(* Schneider Machine Expert - Basic project 29Juli2020, file version 2.4.0.0 *)
(* ProjectInformations: Name=New project *)

HARDWARE
  Cpu 0: TM221CE16R
  ModuleExtensionObject 0: TM3AI8/G
  EthernetConfiguration: NetworkName=M221, IpAllocationMode=FixedAddress, IpAddress=192.168.10.91, SubnetMask=255.255.255.0
  SerialLineConfiguration: Baud=Baud19200, Parity=ParityEven, DataBits=DataBits8, StopBits=StopBits1, PhysicalMedium=PhysicalMediumRs485, TransmissionMode=TransmissionModeModbusRtu, SlaveId=1, Addressing=SlaveAddressing
  MastTask: UsePeriodScanMode=false, PeriodScan=100
  FastTask: Period=255
  CpuBehavior: StartingMode=StartAsPreviousState, AutoSaveRamOnEeprom=true, WatchdogPeriod=250

SYMBOLS  (address, symbol, comment, settings)
  %HSC0       [Type=SimpleCounter, Preset=0, UseDoubleWord=true, DedicatedInputs(DedicatedInput(Activated=true)), ReflexOutputs(ReflexOutput(Activated=false, LessThanS0=false, GreaterOrEqualThanS0=false, GreaterOrEqualThanS1=false), ReflexOutput(Activated=false, LessThanS0=false, GreaterOrEqualThanS0=false, GreaterOrEqualThanS1=false)), Thresholds(Threshold(ThresholdType=NotUsed, Priority=7), Threshold(Threshold]
  %HSC1       [Type=SimpleCounter, Preset=0, UseDoubleWord=true, DedicatedInputs(DedicatedInput(Activated=true)), ReflexOutputs(ReflexOutput(Activated=false, LessThanS0=false, GreaterOrEqualThanS0=false, GreaterOrEqualThanS1=false), ReflexOutput(Activated=false, LessThanS0=false, GreaterOrEqualThanS0=false, GreaterOrEqualThanS1=false)), Thresholds(Threshold(ThresholdType=NotUsed, Priority=7), Threshold(Threshold]
  %IW1.0      [Type=Type_4_20mA, Scope=Scope_Customized, Minimum=4000, Maximum=20000]
  %IW1.1      [Type=Type_4_20mA, Scope=Scope_Customized, Minimum=4000, Maximum=20000]
  %IW1.2      [Type=Type_4_20mA, Scope=Scope_Customized, Minimum=4000, Maximum=20000]
  %IW1.3      [Type=Type_4_20mA, Scope=Scope_Customized, Minimum=4000, Maximum=20000]
  %IW1.4      [Type=Type_4_20mA, Scope=Scope_Customized, Minimum=4000, Maximum=20000]
  %IW1.5      [Type=Type_4_20mA, Scope=Scope_Customized, Minimum=4000, Maximum=20000]
  %IW1.6      [Type=Type_4_20mA, Scope=Scope_Customized, Minimum=4000, Maximum=20000]

POU 4mikronA
  (* SectionNumber=1 *)

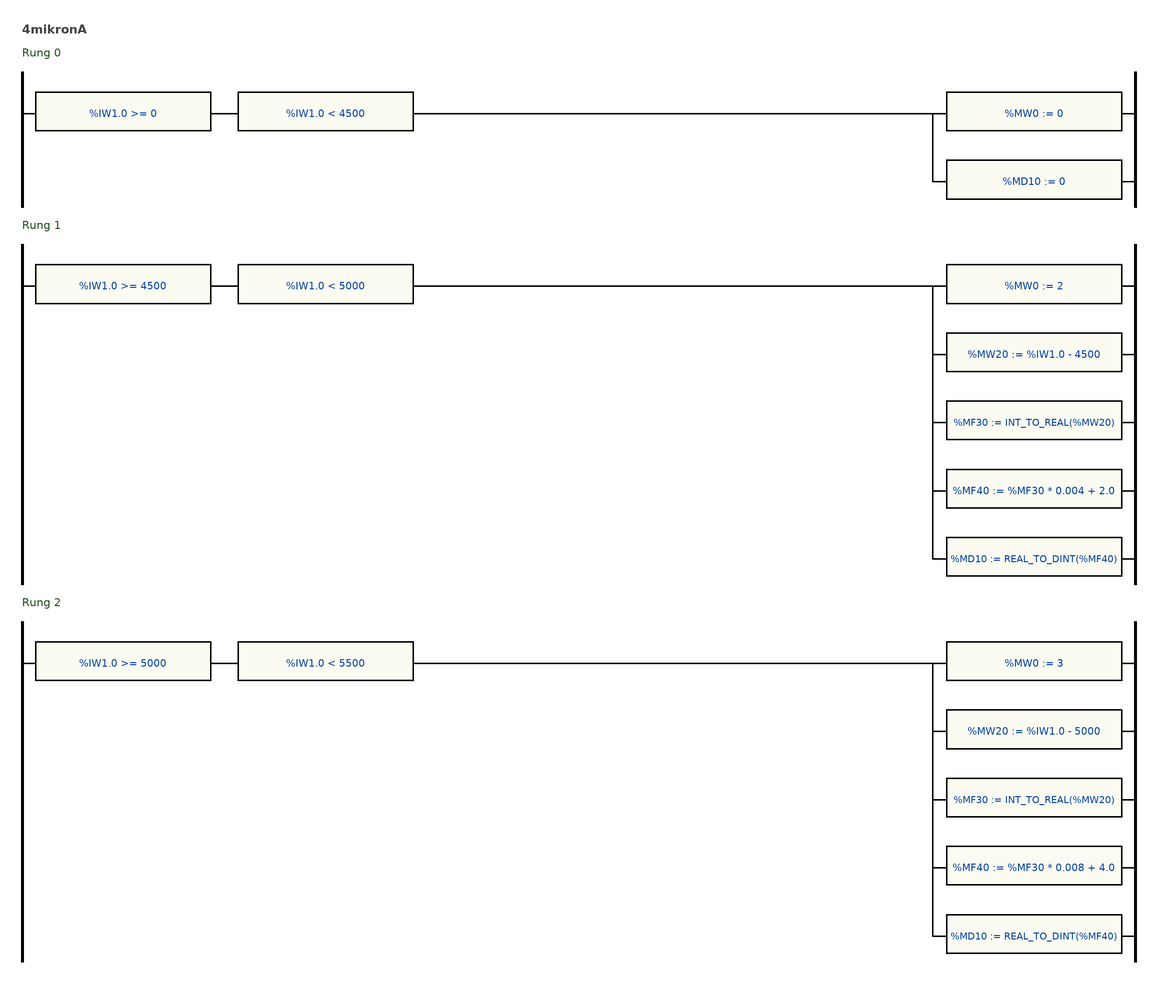

// Rung 0
  LD [ %IW1.0 >= 0 ]
  AND [ %IW1.0 < 4500 ]
  [ %MW0 := 0 ]
  [ %MD10 := 0 ]
  // as ST:
  //   IF %IW1.0 >= 0 AND %IW1.0 < 4500 THEN %MW0 := 0; END_IF;
  //   IF %IW1.0 >= 0 AND %IW1.0 < 4500 THEN %MD10 := 0; END_IF;

// Rung 1
  LD [ %IW1.0 >= 4500 ]
  AND [ %IW1.0 < 5000 ]
  [ %MW0 := 2 ]
  [ %MW20 := %IW1.0 - 4500 ]
  [ %MF30 := INT_TO_REAL ( %MW20 ) ]
  [ %MF40 := %MF30 * 0.004 + 2.0 ]
  [ %MD10 := REAL_TO_DINT ( %MF40 ) ]
  // as ST:
  //   IF %IW1.0 >= 4500 AND %IW1.0 < 5000 THEN %MW0 := 2; END_IF;
  //   IF %IW1.0 >= 4500 AND %IW1.0 < 5000 THEN %MW20 := %IW1.0 - 4500; END_IF;
  //   IF %IW1.0 >= 4500 AND %IW1.0 < 5000 THEN %MF30 := INT_TO_REAL ( %MW20 ); END_IF;
  //   IF %IW1.0 >= 4500 AND %IW1.0 < 5000 THEN %MF40 := %MF30 * 0.004 + 2.0; END_IF;
  //   IF %IW1.0 >= 4500 AND %IW1.0 < 5000 THEN %MD10 := REAL_TO_DINT ( %MF40 ); END_IF;

// Rung 2
  LD [ %IW1.0 >= 5000 ]
  AND [ %IW1.0 < 5500 ]
  [ %MW0 := 3 ]
  [ %MW20 := %IW1.0 - 5000 ]
  [ %MF30 := INT_TO_REAL ( %MW20 ) ]
  [ %MF40 := %MF30 * 0.008 + 4.0 ]
  [ %MD10 := REAL_TO_DINT ( %MF40 ) ]
  // as ST:
  //   IF %IW1.0 >= 5000 AND %IW1.0 < 5500 THEN %MW0 := 3; END_IF;
  //   IF %IW1.0 >= 5000 AND %IW1.0 < 5500 THEN %MW20 := %IW1.0 - 5000; END_IF;
  //   IF %IW1.0 >= 5000 AND %IW1.0 < 5500 THEN %MF30 := INT_TO_REAL ( %MW20 ); END_IF;
  //   IF %IW1.0 >= 5000 AND %IW1.0 < 5500 THEN %MF40 := %MF30 * 0.008 + 4.0; END_IF;
  //   IF %IW1.0 >= 5000 AND %IW1.0 < 5500 THEN %MD10 := REAL_TO_DINT ( %MF40 ); END_IF;

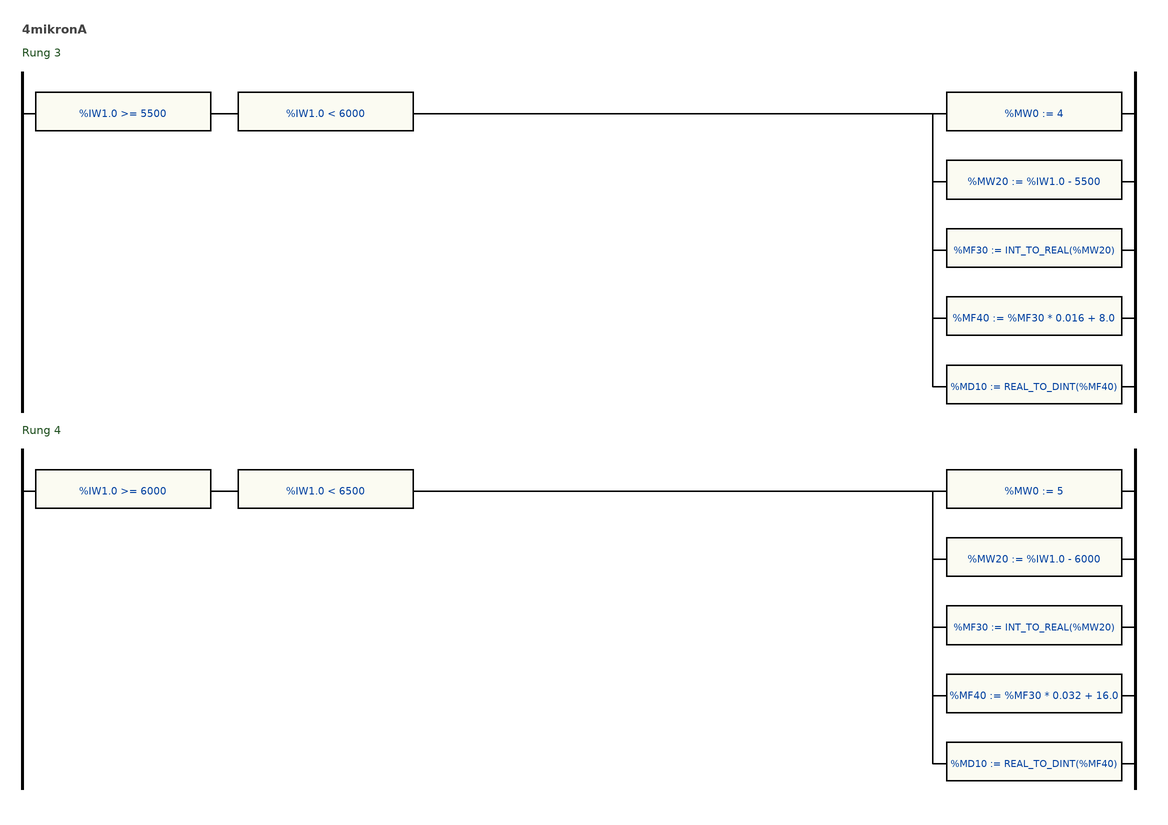

// Rung 3
  LD [ %IW1.0 >= 5500 ]
  AND [ %IW1.0 < 6000 ]
  [ %MW0 := 4 ]
  [ %MW20 := %IW1.0 - 5500 ]
  [ %MF30 := INT_TO_REAL ( %MW20 ) ]
  [ %MF40 := %MF30 * 0.016 + 8.0 ]
  [ %MD10 := REAL_TO_DINT ( %MF40 ) ]
  // as ST:
  //   IF %IW1.0 >= 5500 AND %IW1.0 < 6000 THEN %MW0 := 4; END_IF;
  //   IF %IW1.0 >= 5500 AND %IW1.0 < 6000 THEN %MW20 := %IW1.0 - 5500; END_IF;
  //   IF %IW1.0 >= 5500 AND %IW1.0 < 6000 THEN %MF30 := INT_TO_REAL ( %MW20 ); END_IF;
  //   IF %IW1.0 >= 5500 AND %IW1.0 < 6000 THEN %MF40 := %MF30 * 0.016 + 8.0; END_IF;
  //   IF %IW1.0 >= 5500 AND %IW1.0 < 6000 THEN %MD10 := REAL_TO_DINT ( %MF40 ); END_IF;

// Rung 4
  LD [ %IW1.0 >= 6000 ]
  AND [ %IW1.0 < 6500 ]
  [ %MW0 := 5 ]
  [ %MW20 := %IW1.0 - 6000 ]
  [ %MF30 := INT_TO_REAL ( %MW20 ) ]
  [ %MF40 := %MF30 * 0.032 + 16.0 ]
  [ %MD10 := REAL_TO_DINT ( %MF40 ) ]
  // as ST:
  //   IF %IW1.0 >= 6000 AND %IW1.0 < 6500 THEN %MW0 := 5; END_IF;
  //   IF %IW1.0 >= 6000 AND %IW1.0 < 6500 THEN %MW20 := %IW1.0 - 6000; END_IF;
  //   IF %IW1.0 >= 6000 AND %IW1.0 < 6500 THEN %MF30 := INT_TO_REAL ( %MW20 ); END_IF;
  //   IF %IW1.0 >= 6000 AND %IW1.0 < 6500 THEN %MF40 := %MF30 * 0.032 + 16.0; END_IF;
  //   IF %IW1.0 >= 6000 AND %IW1.0 < 6500 THEN %MD10 := REAL_TO_DINT ( %MF40 ); END_IF;

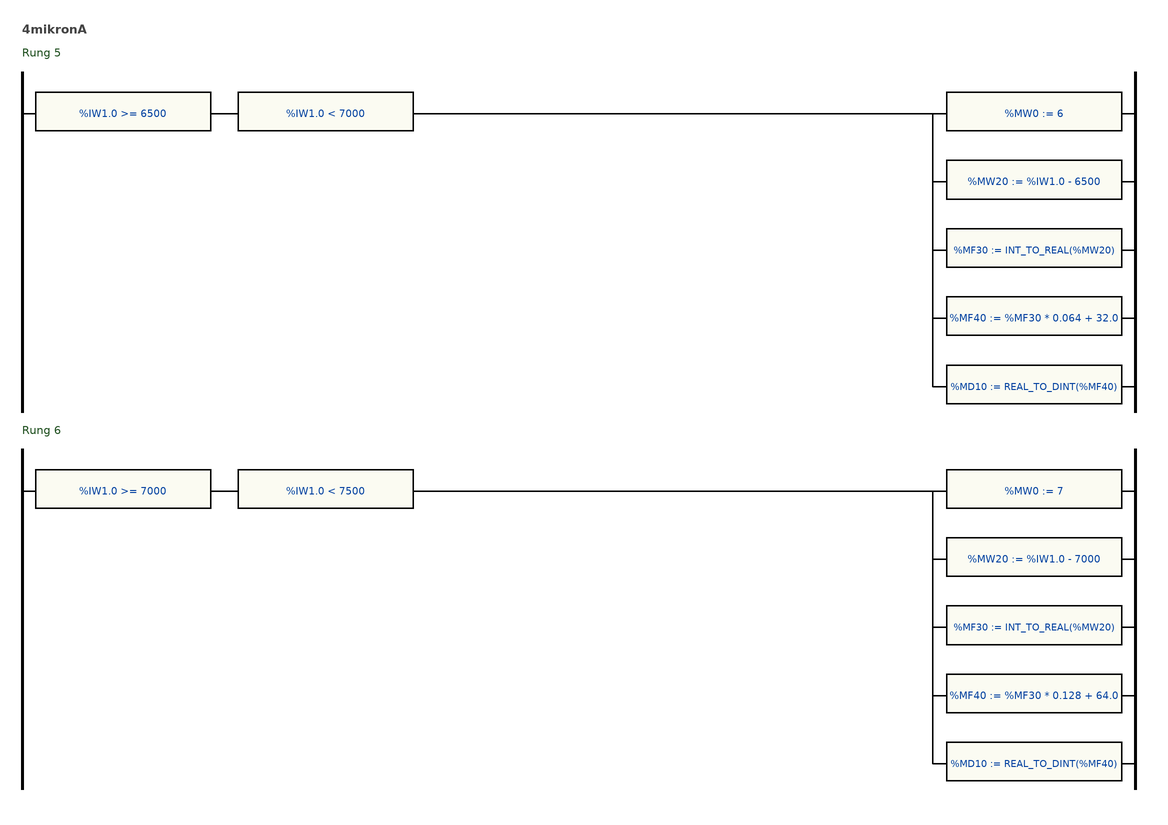

// Rung 5
  LD [ %IW1.0 >= 6500 ]
  AND [ %IW1.0 < 7000 ]
  [ %MW0 := 6 ]
  [ %MW20 := %IW1.0 - 6500 ]
  [ %MF30 := INT_TO_REAL ( %MW20 ) ]
  [ %MF40 := %MF30 * 0.064 + 32.0 ]
  [ %MD10 := REAL_TO_DINT ( %MF40 ) ]
  // as ST:
  //   IF %IW1.0 >= 6500 AND %IW1.0 < 7000 THEN %MW0 := 6; END_IF;
  //   IF %IW1.0 >= 6500 AND %IW1.0 < 7000 THEN %MW20 := %IW1.0 - 6500; END_IF;
  //   IF %IW1.0 >= 6500 AND %IW1.0 < 7000 THEN %MF30 := INT_TO_REAL ( %MW20 ); END_IF;
  //   IF %IW1.0 >= 6500 AND %IW1.0 < 7000 THEN %MF40 := %MF30 * 0.064 + 32.0; END_IF;
  //   IF %IW1.0 >= 6500 AND %IW1.0 < 7000 THEN %MD10 := REAL_TO_DINT ( %MF40 ); END_IF;

// Rung 6
  LD [ %IW1.0 >= 7000 ]
  AND [ %IW1.0 < 7500 ]
  [ %MW0 := 7 ]
  [ %MW20 := %IW1.0 - 7000 ]
  [ %MF30 := INT_TO_REAL ( %MW20 ) ]
  [ %MF40 := %MF30 * 0.128 + 64.0 ]
  [ %MD10 := REAL_TO_DINT ( %MF40 ) ]
  // as ST:
  //   IF %IW1.0 >= 7000 AND %IW1.0 < 7500 THEN %MW0 := 7; END_IF;
  //   IF %IW1.0 >= 7000 AND %IW1.0 < 7500 THEN %MW20 := %IW1.0 - 7000; END_IF;
  //   IF %IW1.0 >= 7000 AND %IW1.0 < 7500 THEN %MF30 := INT_TO_REAL ( %MW20 ); END_IF;
  //   IF %IW1.0 >= 7000 AND %IW1.0 < 7500 THEN %MF40 := %MF30 * 0.128 + 64.0; END_IF;
  //   IF %IW1.0 >= 7000 AND %IW1.0 < 7500 THEN %MD10 := REAL_TO_DINT ( %MF40 ); END_IF;

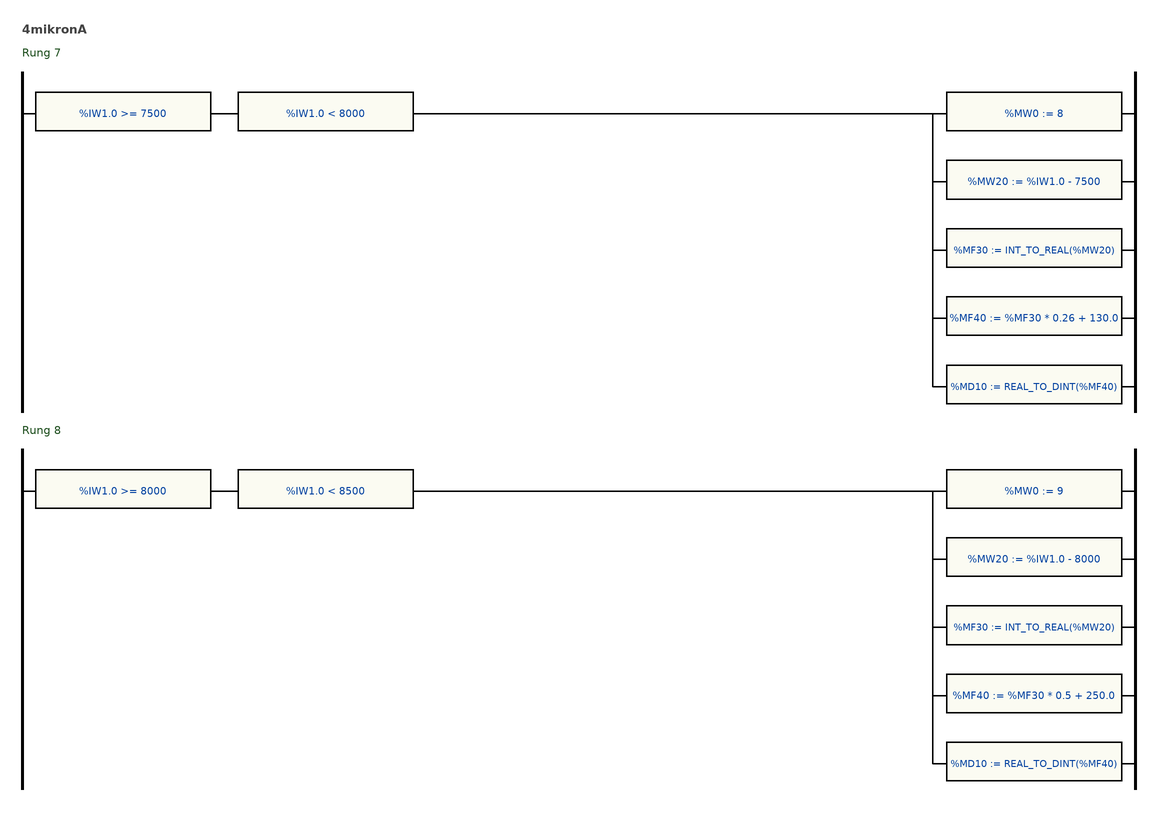

// Rung 7
  LD [ %IW1.0 >= 7500 ]
  AND [ %IW1.0 < 8000 ]
  [ %MW0 := 8 ]
  [ %MW20 := %IW1.0 - 7500 ]
  [ %MF30 := INT_TO_REAL ( %MW20 ) ]
  [ %MF40 := %MF30 * 0.26 + 130.0 ]
  [ %MD10 := REAL_TO_DINT ( %MF40 ) ]
  // as ST:
  //   IF %IW1.0 >= 7500 AND %IW1.0 < 8000 THEN %MW0 := 8; END_IF;
  //   IF %IW1.0 >= 7500 AND %IW1.0 < 8000 THEN %MW20 := %IW1.0 - 7500; END_IF;
  //   IF %IW1.0 >= 7500 AND %IW1.0 < 8000 THEN %MF30 := INT_TO_REAL ( %MW20 ); END_IF;
  //   IF %IW1.0 >= 7500 AND %IW1.0 < 8000 THEN %MF40 := %MF30 * 0.26 + 130.0; END_IF;
  //   IF %IW1.0 >= 7500 AND %IW1.0 < 8000 THEN %MD10 := REAL_TO_DINT ( %MF40 ); END_IF;

// Rung 8
  LD [ %IW1.0 >= 8000 ]
  AND [ %IW1.0 < 8500 ]
  [ %MW0 := 9 ]
  [ %MW20 := %IW1.0 - 8000 ]
  [ %MF30 := INT_TO_REAL ( %MW20 ) ]
  [ %MF40 := %MF30 * 0.5 + 250.0 ]
  [ %MD10 := REAL_TO_DINT ( %MF40 ) ]
  // as ST:
  //   IF %IW1.0 >= 8000 AND %IW1.0 < 8500 THEN %MW0 := 9; END_IF;
  //   IF %IW1.0 >= 8000 AND %IW1.0 < 8500 THEN %MW20 := %IW1.0 - 8000; END_IF;
  //   IF %IW1.0 >= 8000 AND %IW1.0 < 8500 THEN %MF30 := INT_TO_REAL ( %MW20 ); END_IF;
  //   IF %IW1.0 >= 8000 AND %IW1.0 < 8500 THEN %MF40 := %MF30 * 0.5 + 250.0; END_IF;
  //   IF %IW1.0 >= 8000 AND %IW1.0 < 8500 THEN %MD10 := REAL_TO_DINT ( %MF40 ); END_IF;

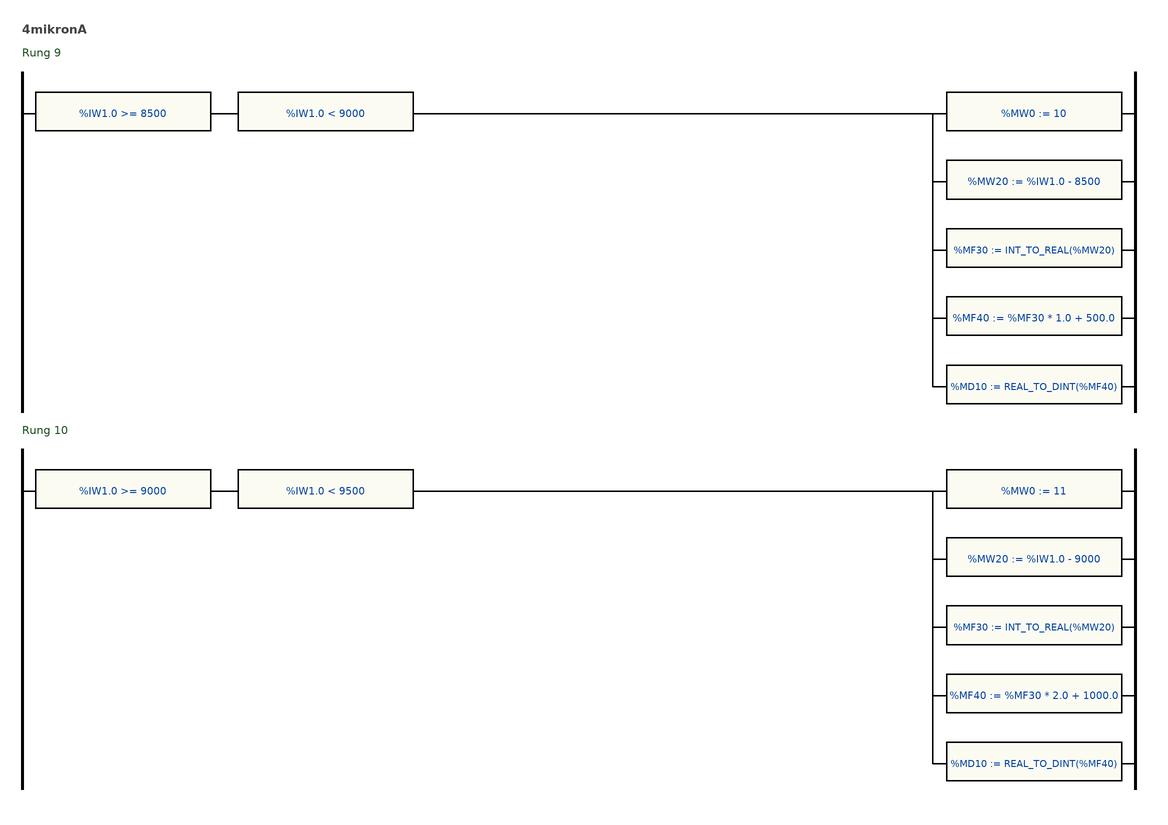

// Rung 9
  LD [ %IW1.0 >= 8500 ]
  AND [ %IW1.0 < 9000 ]
  [ %MW0 := 10 ]
  [ %MW20 := %IW1.0 - 8500 ]
  [ %MF30 := INT_TO_REAL ( %MW20 ) ]
  [ %MF40 := %MF30 * 1.0 + 500.0 ]
  [ %MD10 := REAL_TO_DINT ( %MF40 ) ]
  // as ST:
  //   IF %IW1.0 >= 8500 AND %IW1.0 < 9000 THEN %MW0 := 10; END_IF;
  //   IF %IW1.0 >= 8500 AND %IW1.0 < 9000 THEN %MW20 := %IW1.0 - 8500; END_IF;
  //   IF %IW1.0 >= 8500 AND %IW1.0 < 9000 THEN %MF30 := INT_TO_REAL ( %MW20 ); END_IF;
  //   IF %IW1.0 >= 8500 AND %IW1.0 < 9000 THEN %MF40 := %MF30 * 1.0 + 500.0; END_IF;
  //   IF %IW1.0 >= 8500 AND %IW1.0 < 9000 THEN %MD10 := REAL_TO_DINT ( %MF40 ); END_IF;

// Rung 10
  LD [ %IW1.0 >= 9000 ]
  AND [ %IW1.0 < 9500 ]
  [ %MW0 := 11 ]
  [ %MW20 := %IW1.0 - 9000 ]
  [ %MF30 := INT_TO_REAL ( %MW20 ) ]
  [ %MF40 := %MF30 * 2.0 + 1000.0 ]
  [ %MD10 := REAL_TO_DINT ( %MF40 ) ]
  // as ST:
  //   IF %IW1.0 >= 9000 AND %IW1.0 < 9500 THEN %MW0 := 11; END_IF;
  //   IF %IW1.0 >= 9000 AND %IW1.0 < 9500 THEN %MW20 := %IW1.0 - 9000; END_IF;
  //   IF %IW1.0 >= 9000 AND %IW1.0 < 9500 THEN %MF30 := INT_TO_REAL ( %MW20 ); END_IF;
  //   IF %IW1.0 >= 9000 AND %IW1.0 < 9500 THEN %MF40 := %MF30 * 2.0 + 1000.0; END_IF;
  //   IF %IW1.0 >= 9000 AND %IW1.0 < 9500 THEN %MD10 := REAL_TO_DINT ( %MF40 ); END_IF;

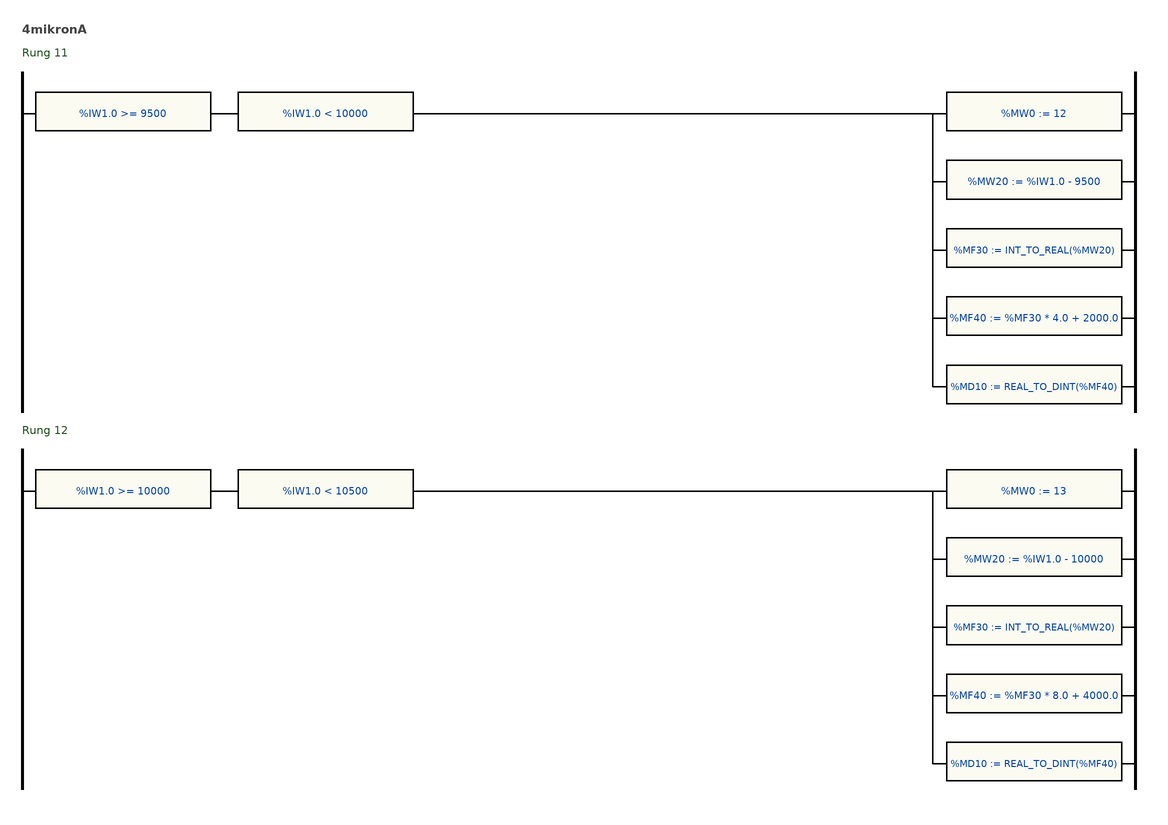

// Rung 11
  LD [ %IW1.0 >= 9500 ]
  AND [ %IW1.0 < 10000 ]
  [ %MW0 := 12 ]
  [ %MW20 := %IW1.0 - 9500 ]
  [ %MF30 := INT_TO_REAL ( %MW20 ) ]
  [ %MF40 := %MF30 * 4.0 + 2000.0 ]
  [ %MD10 := REAL_TO_DINT ( %MF40 ) ]
  // as ST:
  //   IF %IW1.0 >= 9500 AND %IW1.0 < 10000 THEN %MW0 := 12; END_IF;
  //   IF %IW1.0 >= 9500 AND %IW1.0 < 10000 THEN %MW20 := %IW1.0 - 9500; END_IF;
  //   IF %IW1.0 >= 9500 AND %IW1.0 < 10000 THEN %MF30 := INT_TO_REAL ( %MW20 ); END_IF;
  //   IF %IW1.0 >= 9500 AND %IW1.0 < 10000 THEN %MF40 := %MF30 * 4.0 + 2000.0; END_IF;
  //   IF %IW1.0 >= 9500 AND %IW1.0 < 10000 THEN %MD10 := REAL_TO_DINT ( %MF40 ); END_IF;

// Rung 12
  LD [ %IW1.0 >= 10000 ]
  AND [ %IW1.0 < 10500 ]
  [ %MW0 := 13 ]
  [ %MW20 := %IW1.0 - 10000 ]
  [ %MF30 := INT_TO_REAL ( %MW20 ) ]
  [ %MF40 := %MF30 * 8.0 + 4000.0 ]
  [ %MD10 := REAL_TO_DINT ( %MF40 ) ]
  // as ST:
  //   IF %IW1.0 >= 10000 AND %IW1.0 < 10500 THEN %MW0 := 13; END_IF;
  //   IF %IW1.0 >= 10000 AND %IW1.0 < 10500 THEN %MW20 := %IW1.0 - 10000; END_IF;
  //   IF %IW1.0 >= 10000 AND %IW1.0 < 10500 THEN %MF30 := INT_TO_REAL ( %MW20 ); END_IF;
  //   IF %IW1.0 >= 10000 AND %IW1.0 < 10500 THEN %MF40 := %MF30 * 8.0 + 4000.0; END_IF;
  //   IF %IW1.0 >= 10000 AND %IW1.0 < 10500 THEN %MD10 := REAL_TO_DINT ( %MF40 ); END_IF;

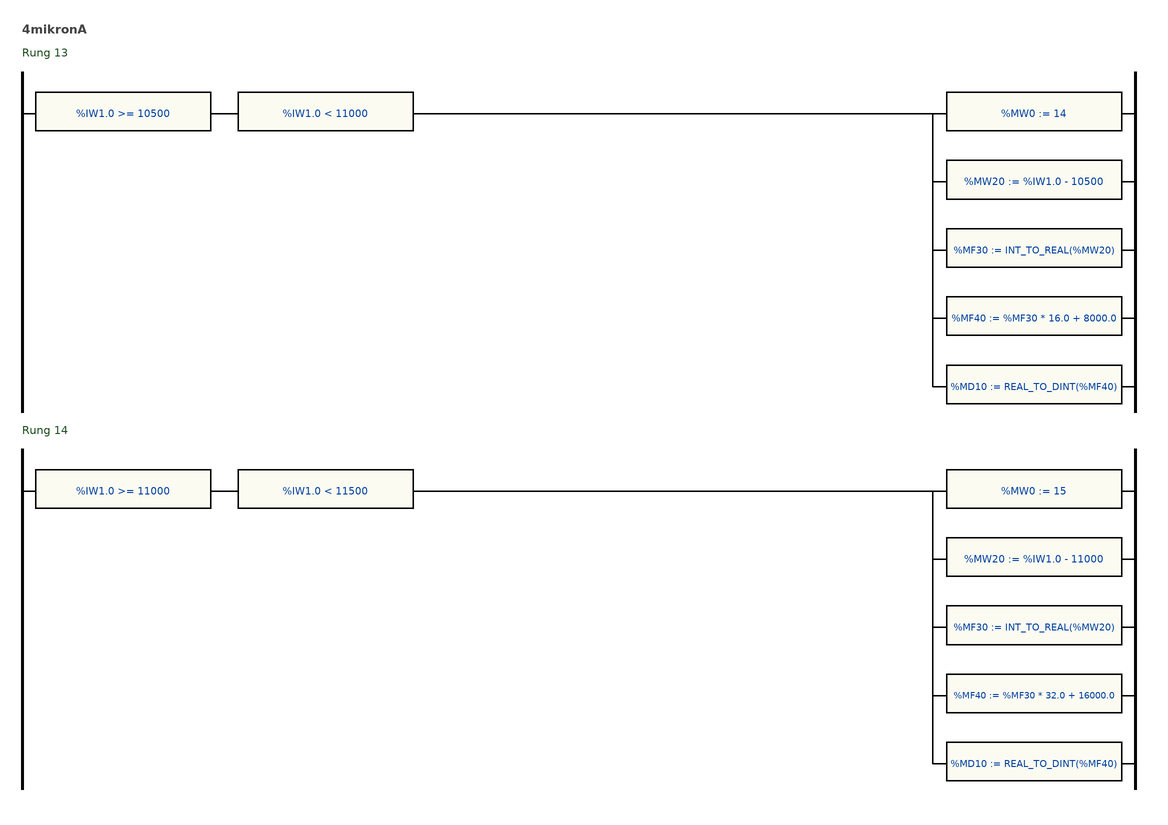

// Rung 13
  LD [ %IW1.0 >= 10500 ]
  AND [ %IW1.0 < 11000 ]
  [ %MW0 := 14 ]
  [ %MW20 := %IW1.0 - 10500 ]
  [ %MF30 := INT_TO_REAL ( %MW20 ) ]
  [ %MF40 := %MF30 * 16.0 + 8000.0 ]
  [ %MD10 := REAL_TO_DINT ( %MF40 ) ]
  // as ST:
  //   IF %IW1.0 >= 10500 AND %IW1.0 < 11000 THEN %MW0 := 14; END_IF;
  //   IF %IW1.0 >= 10500 AND %IW1.0 < 11000 THEN %MW20 := %IW1.0 - 10500; END_IF;
  //   IF %IW1.0 >= 10500 AND %IW1.0 < 11000 THEN %MF30 := INT_TO_REAL ( %MW20 ); END_IF;
  //   IF %IW1.0 >= 10500 AND %IW1.0 < 11000 THEN %MF40 := %MF30 * 16.0 + 8000.0; END_IF;
  //   IF %IW1.0 >= 10500 AND %IW1.0 < 11000 THEN %MD10 := REAL_TO_DINT ( %MF40 ); END_IF;

// Rung 14
  LD [ %IW1.0 >= 11000 ]
  AND [ %IW1.0 < 11500 ]
  [ %MW0 := 15 ]
  [ %MW20 := %IW1.0 - 11000 ]
  [ %MF30 := INT_TO_REAL ( %MW20 ) ]
  [ %MF40 := %MF30 * 32.0 + 16000.0 ]
  [ %MD10 := REAL_TO_DINT ( %MF40 ) ]
  // as ST:
  //   IF %IW1.0 >= 11000 AND %IW1.0 < 11500 THEN %MW0 := 15; END_IF;
  //   IF %IW1.0 >= 11000 AND %IW1.0 < 11500 THEN %MW20 := %IW1.0 - 11000; END_IF;
  //   IF %IW1.0 >= 11000 AND %IW1.0 < 11500 THEN %MF30 := INT_TO_REAL ( %MW20 ); END_IF;
  //   IF %IW1.0 >= 11000 AND %IW1.0 < 11500 THEN %MF40 := %MF30 * 32.0 + 16000.0; END_IF;
  //   IF %IW1.0 >= 11000 AND %IW1.0 < 11500 THEN %MD10 := REAL_TO_DINT ( %MF40 ); END_IF;

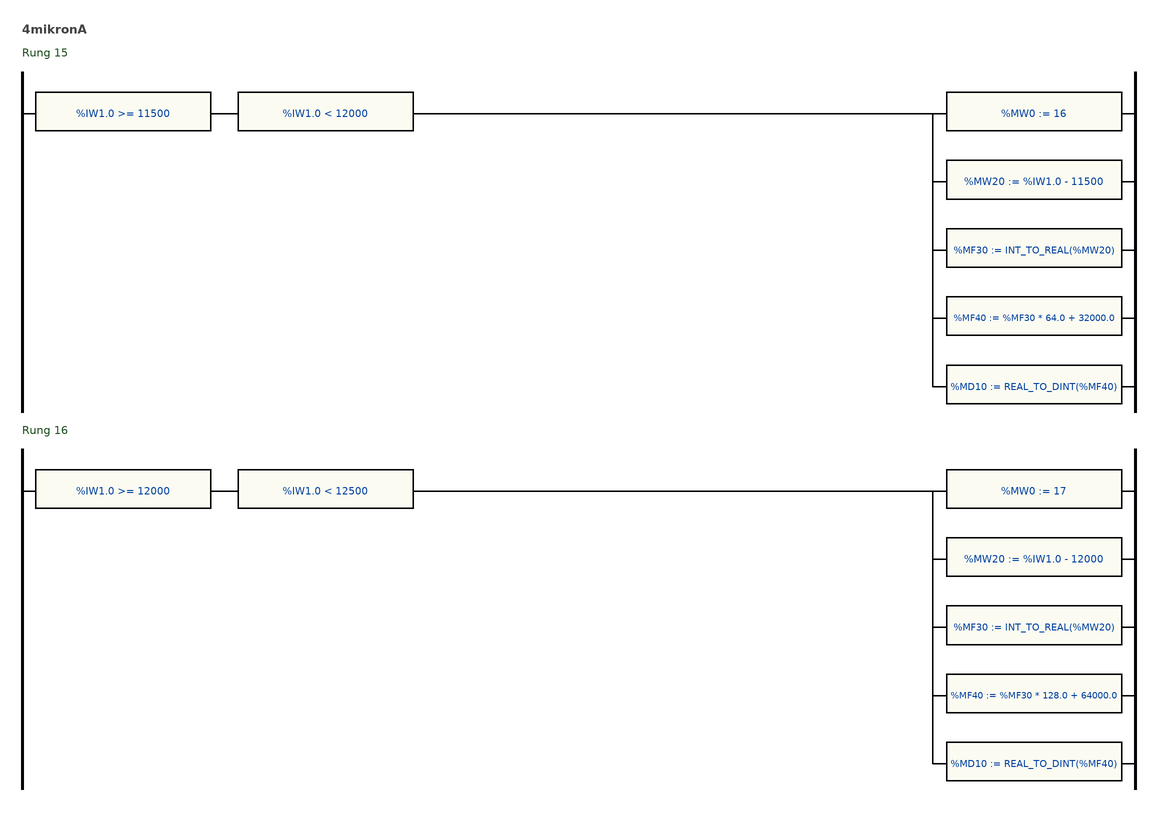

// Rung 15
  LD [ %IW1.0 >= 11500 ]
  AND [ %IW1.0 < 12000 ]
  [ %MW0 := 16 ]
  [ %MW20 := %IW1.0 - 11500 ]
  [ %MF30 := INT_TO_REAL ( %MW20 ) ]
  [ %MF40 := %MF30 * 64.0 + 32000.0 ]
  [ %MD10 := REAL_TO_DINT ( %MF40 ) ]
  // as ST:
  //   IF %IW1.0 >= 11500 AND %IW1.0 < 12000 THEN %MW0 := 16; END_IF;
  //   IF %IW1.0 >= 11500 AND %IW1.0 < 12000 THEN %MW20 := %IW1.0 - 11500; END_IF;
  //   IF %IW1.0 >= 11500 AND %IW1.0 < 12000 THEN %MF30 := INT_TO_REAL ( %MW20 ); END_IF;
  //   IF %IW1.0 >= 11500 AND %IW1.0 < 12000 THEN %MF40 := %MF30 * 64.0 + 32000.0; END_IF;
  //   IF %IW1.0 >= 11500 AND %IW1.0 < 12000 THEN %MD10 := REAL_TO_DINT ( %MF40 ); END_IF;

// Rung 16
  LD [ %IW1.0 >= 12000 ]
  AND [ %IW1.0 < 12500 ]
  [ %MW0 := 17 ]
  [ %MW20 := %IW1.0 - 12000 ]
  [ %MF30 := INT_TO_REAL ( %MW20 ) ]
  [ %MF40 := %MF30 * 128.0 + 64000.0 ]
  [ %MD10 := REAL_TO_DINT ( %MF40 ) ]
  // as ST:
  //   IF %IW1.0 >= 12000 AND %IW1.0 < 12500 THEN %MW0 := 17; END_IF;
  //   IF %IW1.0 >= 12000 AND %IW1.0 < 12500 THEN %MW20 := %IW1.0 - 12000; END_IF;
  //   IF %IW1.0 >= 12000 AND %IW1.0 < 12500 THEN %MF30 := INT_TO_REAL ( %MW20 ); END_IF;
  //   IF %IW1.0 >= 12000 AND %IW1.0 < 12500 THEN %MF40 := %MF30 * 128.0 + 64000.0; END_IF;
  //   IF %IW1.0 >= 12000 AND %IW1.0 < 12500 THEN %MD10 := REAL_TO_DINT ( %MF40 ); END_IF;

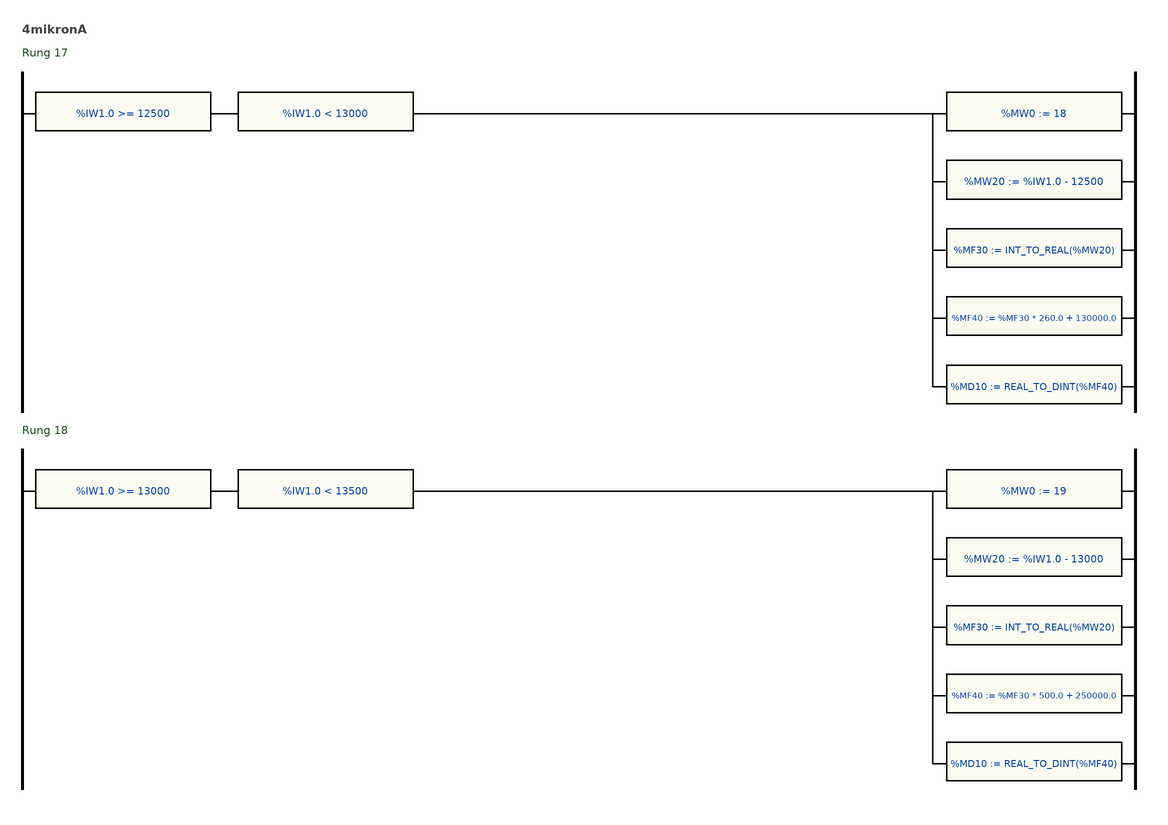

// Rung 17
  LD [ %IW1.0 >= 12500 ]
  AND [ %IW1.0 < 13000 ]
  [ %MW0 := 18 ]
  [ %MW20 := %IW1.0 - 12500 ]
  [ %MF30 := INT_TO_REAL ( %MW20 ) ]
  [ %MF40 := %MF30 * 260.0 + 130000.0 ]
  [ %MD10 := REAL_TO_DINT ( %MF40 ) ]
  // as ST:
  //   IF %IW1.0 >= 12500 AND %IW1.0 < 13000 THEN %MW0 := 18; END_IF;
  //   IF %IW1.0 >= 12500 AND %IW1.0 < 13000 THEN %MW20 := %IW1.0 - 12500; END_IF;
  //   IF %IW1.0 >= 12500 AND %IW1.0 < 13000 THEN %MF30 := INT_TO_REAL ( %MW20 ); END_IF;
  //   IF %IW1.0 >= 12500 AND %IW1.0 < 13000 THEN %MF40 := %MF30 * 260.0 + 130000.0; END_IF;
  //   IF %IW1.0 >= 12500 AND %IW1.0 < 13000 THEN %MD10 := REAL_TO_DINT ( %MF40 ); END_IF;

// Rung 18
  LD [ %IW1.0 >= 13000 ]
  AND [ %IW1.0 < 13500 ]
  [ %MW0 := 19 ]
  [ %MW20 := %IW1.0 - 13000 ]
  [ %MF30 := INT_TO_REAL ( %MW20 ) ]
  [ %MF40 := %MF30 * 500.0 + 250000.0 ]
  [ %MD10 := REAL_TO_DINT ( %MF40 ) ]
  // as ST:
  //   IF %IW1.0 >= 13000 AND %IW1.0 < 13500 THEN %MW0 := 19; END_IF;
  //   IF %IW1.0 >= 13000 AND %IW1.0 < 13500 THEN %MW20 := %IW1.0 - 13000; END_IF;
  //   IF %IW1.0 >= 13000 AND %IW1.0 < 13500 THEN %MF30 := INT_TO_REAL ( %MW20 ); END_IF;
  //   IF %IW1.0 >= 13000 AND %IW1.0 < 13500 THEN %MF40 := %MF30 * 500.0 + 250000.0; END_IF;
  //   IF %IW1.0 >= 13000 AND %IW1.0 < 13500 THEN %MD10 := REAL_TO_DINT ( %MF40 ); END_IF;

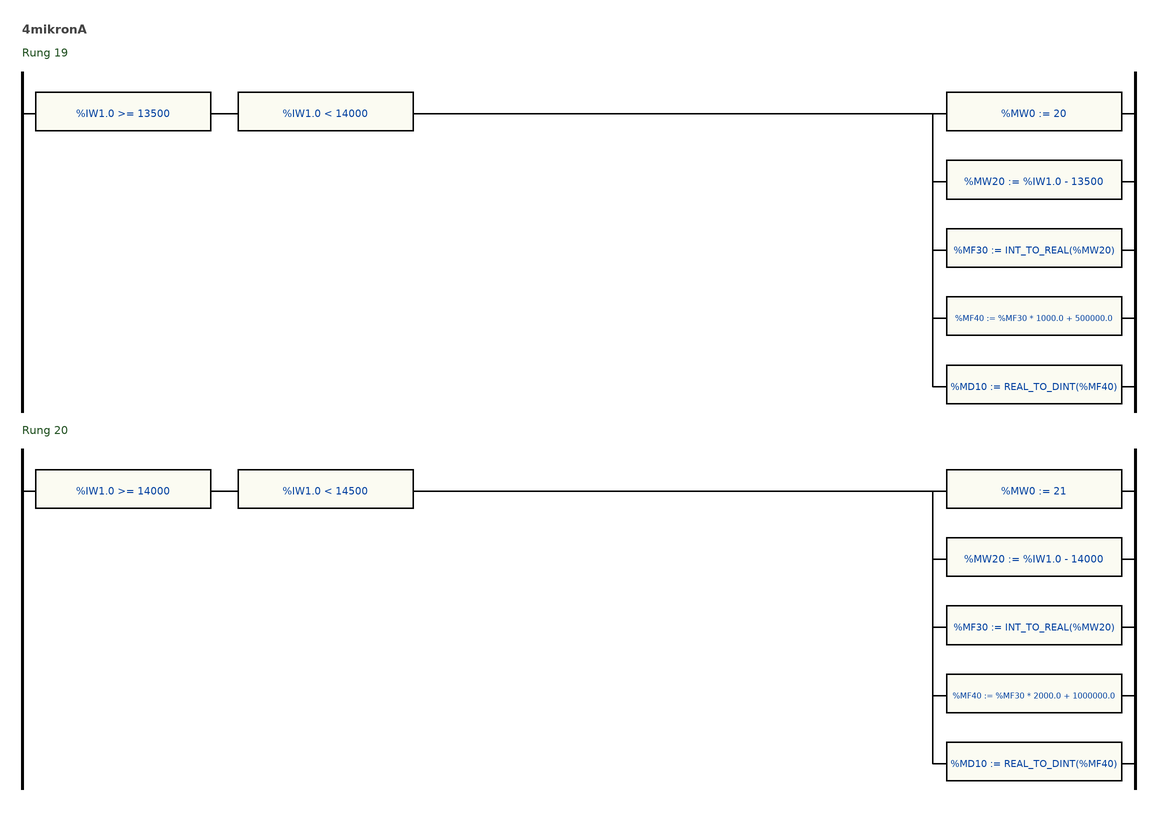

// Rung 19
  LD [ %IW1.0 >= 13500 ]
  AND [ %IW1.0 < 14000 ]
  [ %MW0 := 20 ]
  [ %MW20 := %IW1.0 - 13500 ]
  [ %MF30 := INT_TO_REAL ( %MW20 ) ]
  [ %MF40 := %MF30 * 1000.0 + 500000.0 ]
  [ %MD10 := REAL_TO_DINT ( %MF40 ) ]
  // as ST:
  //   IF %IW1.0 >= 13500 AND %IW1.0 < 14000 THEN %MW0 := 20; END_IF;
  //   IF %IW1.0 >= 13500 AND %IW1.0 < 14000 THEN %MW20 := %IW1.0 - 13500; END_IF;
  //   IF %IW1.0 >= 13500 AND %IW1.0 < 14000 THEN %MF30 := INT_TO_REAL ( %MW20 ); END_IF;
  //   IF %IW1.0 >= 13500 AND %IW1.0 < 14000 THEN %MF40 := %MF30 * 1000.0 + 500000.0; END_IF;
  //   IF %IW1.0 >= 13500 AND %IW1.0 < 14000 THEN %MD10 := REAL_TO_DINT ( %MF40 ); END_IF;

// Rung 20
  LD [ %IW1.0 >= 14000 ]
  AND [ %IW1.0 < 14500 ]
  [ %MW0 := 21 ]
  [ %MW20 := %IW1.0 - 14000 ]
  [ %MF30 := INT_TO_REAL ( %MW20 ) ]
  [ %MF40 := %MF30 * 2000.0 + 1000000.0 ]
  [ %MD10 := REAL_TO_DINT ( %MF40 ) ]
  // as ST:
  //   IF %IW1.0 >= 14000 AND %IW1.0 < 14500 THEN %MW0 := 21; END_IF;
  //   IF %IW1.0 >= 14000 AND %IW1.0 < 14500 THEN %MW20 := %IW1.0 - 14000; END_IF;
  //   IF %IW1.0 >= 14000 AND %IW1.0 < 14500 THEN %MF30 := INT_TO_REAL ( %MW20 ); END_IF;
  //   IF %IW1.0 >= 14000 AND %IW1.0 < 14500 THEN %MF40 := %MF30 * 2000.0 + 1000000.0; END_IF;
  //   IF %IW1.0 >= 14000 AND %IW1.0 < 14500 THEN %MD10 := REAL_TO_DINT ( %MF40 ); END_IF;

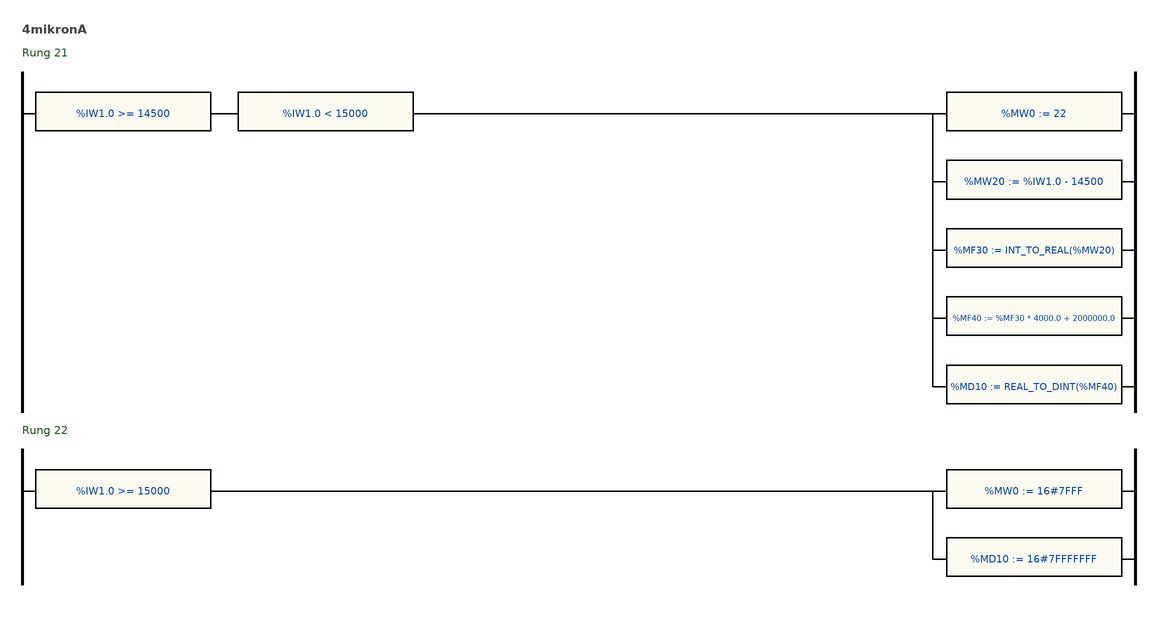

// Rung 21
  LD [ %IW1.0 >= 14500 ]
  AND [ %IW1.0 < 15000 ]
  [ %MW0 := 22 ]
  [ %MW20 := %IW1.0 - 14500 ]
  [ %MF30 := INT_TO_REAL ( %MW20 ) ]
  [ %MF40 := %MF30 * 4000.0 + 2000000.0 ]
  [ %MD10 := REAL_TO_DINT ( %MF40 ) ]
  // as ST:
  //   IF %IW1.0 >= 14500 AND %IW1.0 < 15000 THEN %MW0 := 22; END_IF;
  //   IF %IW1.0 >= 14500 AND %IW1.0 < 15000 THEN %MW20 := %IW1.0 - 14500; END_IF;
  //   IF %IW1.0 >= 14500 AND %IW1.0 < 15000 THEN %MF30 := INT_TO_REAL ( %MW20 ); END_IF;
  //   IF %IW1.0 >= 14500 AND %IW1.0 < 15000 THEN %MF40 := %MF30 * 4000.0 + 2000000.0; END_IF;
  //   IF %IW1.0 >= 14500 AND %IW1.0 < 15000 THEN %MD10 := REAL_TO_DINT ( %MF40 ); END_IF;

// Rung 22
  LD [ %IW1.0 >= 15000 ]
  [ %MW0 := 16#7FFF ]
  [ %MD10 := 16#7FFFFFFF ]
  // as ST:
  //   IF %IW1.0 >= 15000 THEN %MW0 := 16#7FFF; END_IF;
  //   IF %IW1.0 >= 15000 THEN %MD10 := 16#7FFFFFFF; END_IF;

POU 6mikronA
  (* SectionNumber=2 *)

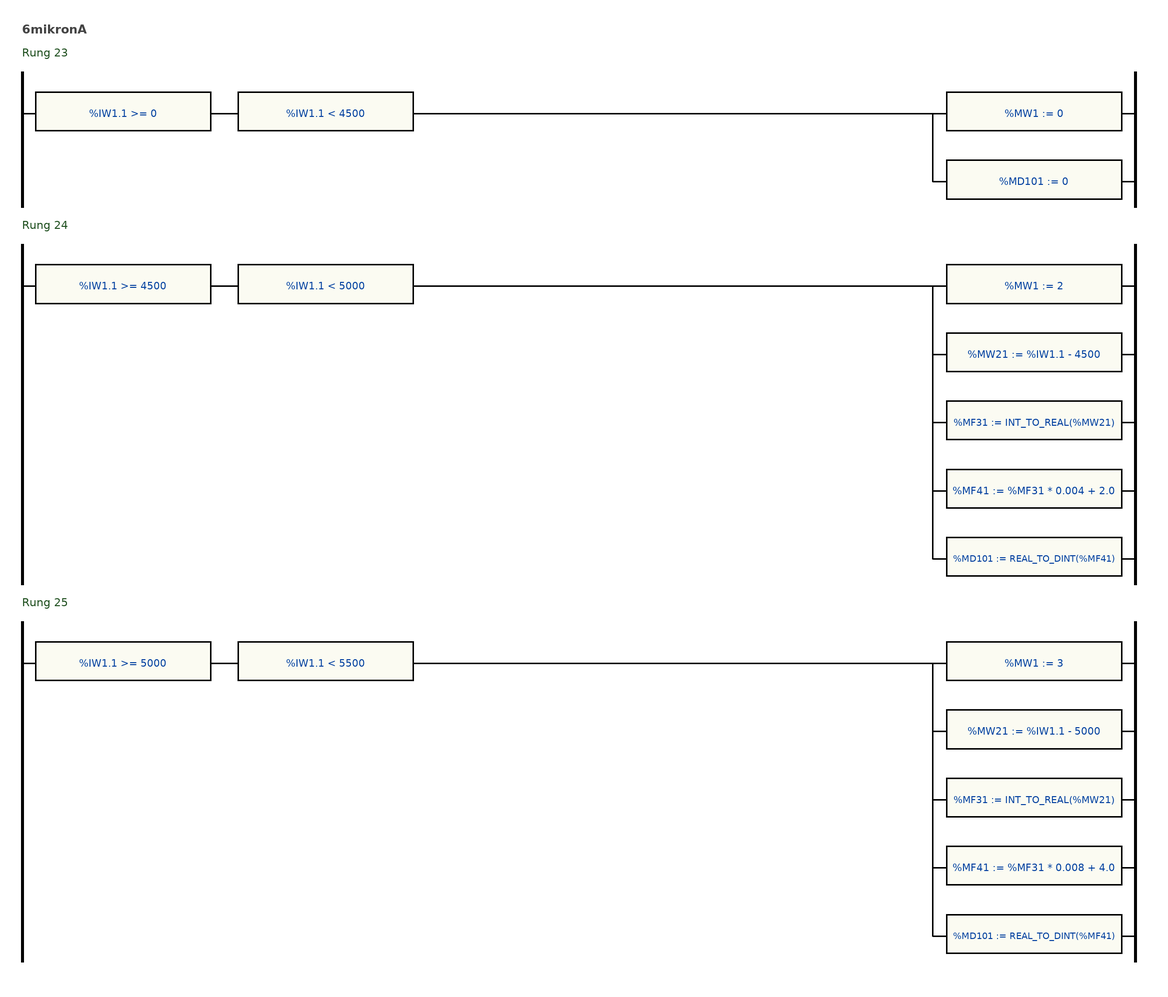

// Rung 23
  LD [ %IW1.1 >= 0 ]
  AND [ %IW1.1 < 4500 ]
  [ %MW1 := 0 ]
  [ %MD101 := 0 ]
  // as ST:
  //   IF %IW1.1 >= 0 AND %IW1.1 < 4500 THEN %MW1 := 0; END_IF;
  //   IF %IW1.1 >= 0 AND %IW1.1 < 4500 THEN %MD101 := 0; END_IF;

// Rung 24
  LD [ %IW1.1 >= 4500 ]
  AND [ %IW1.1 < 5000 ]
  [ %MW1 := 2 ]
  [ %MW21 := %IW1.1 - 4500 ]
  [ %MF31 := INT_TO_REAL ( %MW21 ) ]
  [ %MF41 := %MF31 * 0.004 + 2.0 ]
  [ %MD101 := REAL_TO_DINT ( %MF41 ) ]
  // as ST:
  //   IF %IW1.1 >= 4500 AND %IW1.1 < 5000 THEN %MW1 := 2; END_IF;
  //   IF %IW1.1 >= 4500 AND %IW1.1 < 5000 THEN %MW21 := %IW1.1 - 4500; END_IF;
  //   IF %IW1.1 >= 4500 AND %IW1.1 < 5000 THEN %MF31 := INT_TO_REAL ( %MW21 ); END_IF;
  //   IF %IW1.1 >= 4500 AND %IW1.1 < 5000 THEN %MF41 := %MF31 * 0.004 + 2.0; END_IF;
  //   IF %IW1.1 >= 4500 AND %IW1.1 < 5000 THEN %MD101 := REAL_TO_DINT ( %MF41 ); END_IF;

// Rung 25
  LD [ %IW1.1 >= 5000 ]
  AND [ %IW1.1 < 5500 ]
  [ %MW1 := 3 ]
  [ %MW21 := %IW1.1 - 5000 ]
  [ %MF31 := INT_TO_REAL ( %MW21 ) ]
  [ %MF41 := %MF31 * 0.008 + 4.0 ]
  [ %MD101 := REAL_TO_DINT ( %MF41 ) ]
  // as ST:
  //   IF %IW1.1 >= 5000 AND %IW1.1 < 5500 THEN %MW1 := 3; END_IF;
  //   IF %IW1.1 >= 5000 AND %IW1.1 < 5500 THEN %MW21 := %IW1.1 - 5000; END_IF;
  //   IF %IW1.1 >= 5000 AND %IW1.1 < 5500 THEN %MF31 := INT_TO_REAL ( %MW21 ); END_IF;
  //   IF %IW1.1 >= 5000 AND %IW1.1 < 5500 THEN %MF41 := %MF31 * 0.008 + 4.0; END_IF;
  //   IF %IW1.1 >= 5000 AND %IW1.1 < 5500 THEN %MD101 := REAL_TO_DINT ( %MF41 ); END_IF;

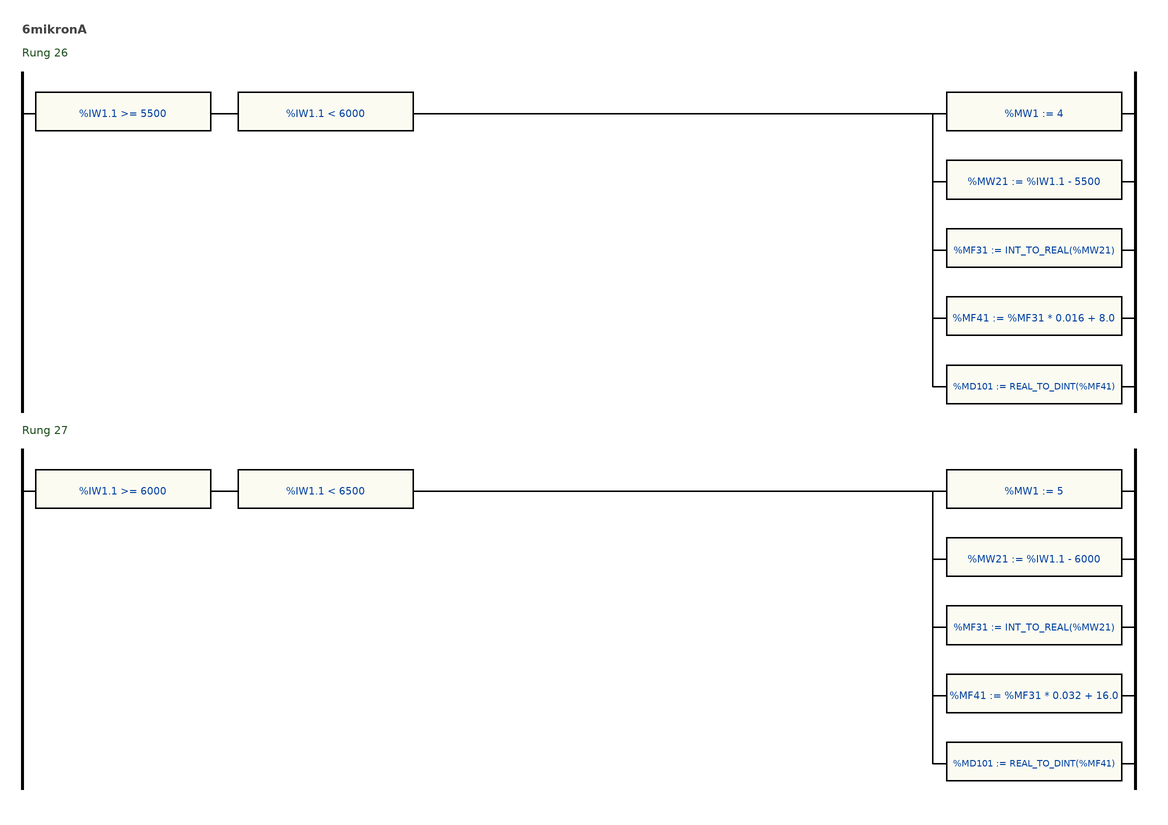

// Rung 26
  LD [ %IW1.1 >= 5500 ]
  AND [ %IW1.1 < 6000 ]
  [ %MW1 := 4 ]
  [ %MW21 := %IW1.1 - 5500 ]
  [ %MF31 := INT_TO_REAL ( %MW21 ) ]
  [ %MF41 := %MF31 * 0.016 + 8.0 ]
  [ %MD101 := REAL_TO_DINT ( %MF41 ) ]
  // as ST:
  //   IF %IW1.1 >= 5500 AND %IW1.1 < 6000 THEN %MW1 := 4; END_IF;
  //   IF %IW1.1 >= 5500 AND %IW1.1 < 6000 THEN %MW21 := %IW1.1 - 5500; END_IF;
  //   IF %IW1.1 >= 5500 AND %IW1.1 < 6000 THEN %MF31 := INT_TO_REAL ( %MW21 ); END_IF;
  //   IF %IW1.1 >= 5500 AND %IW1.1 < 6000 THEN %MF41 := %MF31 * 0.016 + 8.0; END_IF;
  //   IF %IW1.1 >= 5500 AND %IW1.1 < 6000 THEN %MD101 := REAL_TO_DINT ( %MF41 ); END_IF;

// Rung 27
  LD [ %IW1.1 >= 6000 ]
  AND [ %IW1.1 < 6500 ]
  [ %MW1 := 5 ]
  [ %MW21 := %IW1.1 - 6000 ]
  [ %MF31 := INT_TO_REAL ( %MW21 ) ]
  [ %MF41 := %MF31 * 0.032 + 16.0 ]
  [ %MD101 := REAL_TO_DINT ( %MF41 ) ]
  // as ST:
  //   IF %IW1.1 >= 6000 AND %IW1.1 < 6500 THEN %MW1 := 5; END_IF;
  //   IF %IW1.1 >= 6000 AND %IW1.1 < 6500 THEN %MW21 := %IW1.1 - 6000; END_IF;
  //   IF %IW1.1 >= 6000 AND %IW1.1 < 6500 THEN %MF31 := INT_TO_REAL ( %MW21 ); END_IF;
  //   IF %IW1.1 >= 6000 AND %IW1.1 < 6500 THEN %MF41 := %MF31 * 0.032 + 16.0; END_IF;
  //   IF %IW1.1 >= 6000 AND %IW1.1 < 6500 THEN %MD101 := REAL_TO_DINT ( %MF41 ); END_IF;

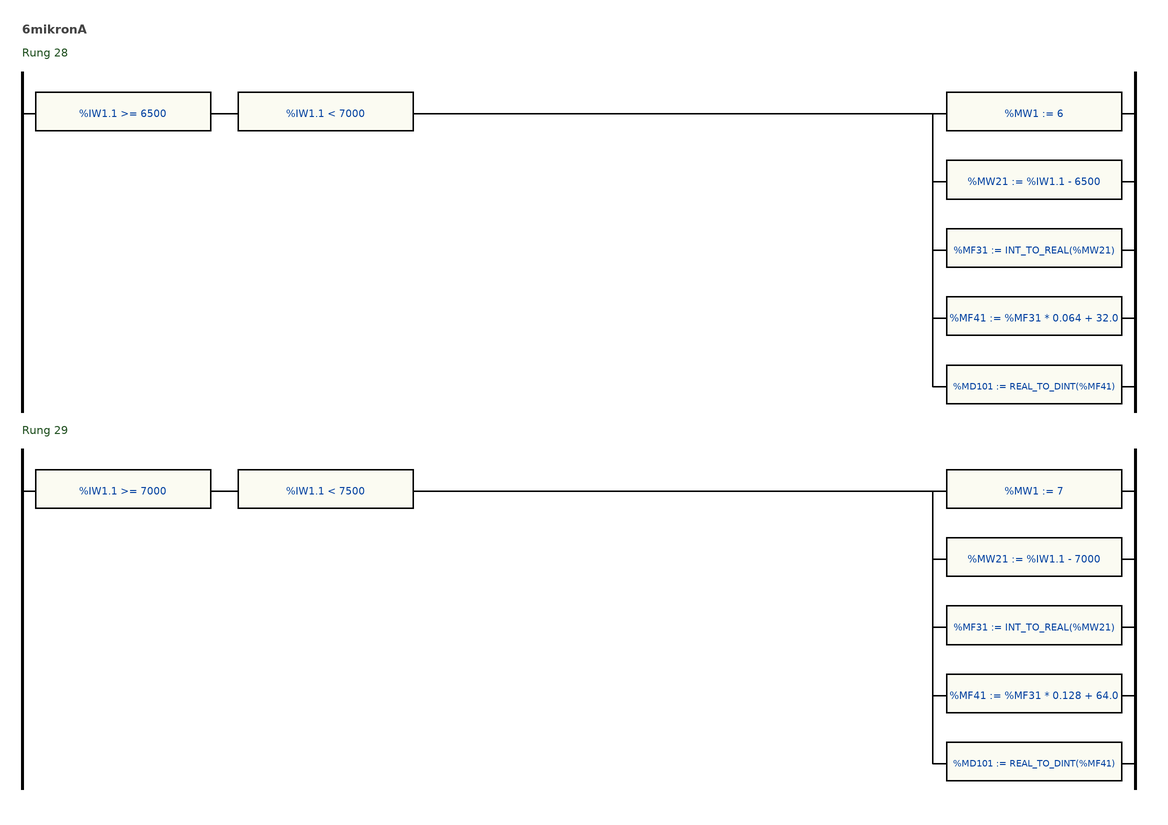

// Rung 28
  LD [ %IW1.1 >= 6500 ]
  AND [ %IW1.1 < 7000 ]
  [ %MW1 := 6 ]
  [ %MW21 := %IW1.1 - 6500 ]
  [ %MF31 := INT_TO_REAL ( %MW21 ) ]
  [ %MF41 := %MF31 * 0.064 + 32.0 ]
  [ %MD101 := REAL_TO_DINT ( %MF41 ) ]
  // as ST:
  //   IF %IW1.1 >= 6500 AND %IW1.1 < 7000 THEN %MW1 := 6; END_IF;
  //   IF %IW1.1 >= 6500 AND %IW1.1 < 7000 THEN %MW21 := %IW1.1 - 6500; END_IF;
  //   IF %IW1.1 >= 6500 AND %IW1.1 < 7000 THEN %MF31 := INT_TO_REAL ( %MW21 ); END_IF;
  //   IF %IW1.1 >= 6500 AND %IW1.1 < 7000 THEN %MF41 := %MF31 * 0.064 + 32.0; END_IF;
  //   IF %IW1.1 >= 6500 AND %IW1.1 < 7000 THEN %MD101 := REAL_TO_DINT ( %MF41 ); END_IF;

// Rung 29
  LD [ %IW1.1 >= 7000 ]
  AND [ %IW1.1 < 7500 ]
  [ %MW1 := 7 ]
  [ %MW21 := %IW1.1 - 7000 ]
  [ %MF31 := INT_TO_REAL ( %MW21 ) ]
  [ %MF41 := %MF31 * 0.128 + 64.0 ]
  [ %MD101 := REAL_TO_DINT ( %MF41 ) ]
  // as ST:
  //   IF %IW1.1 >= 7000 AND %IW1.1 < 7500 THEN %MW1 := 7; END_IF;
  //   IF %IW1.1 >= 7000 AND %IW1.1 < 7500 THEN %MW21 := %IW1.1 - 7000; END_IF;
  //   IF %IW1.1 >= 7000 AND %IW1.1 < 7500 THEN %MF31 := INT_TO_REAL ( %MW21 ); END_IF;
  //   IF %IW1.1 >= 7000 AND %IW1.1 < 7500 THEN %MF41 := %MF31 * 0.128 + 64.0; END_IF;
  //   IF %IW1.1 >= 7000 AND %IW1.1 < 7500 THEN %MD101 := REAL_TO_DINT ( %MF41 ); END_IF;

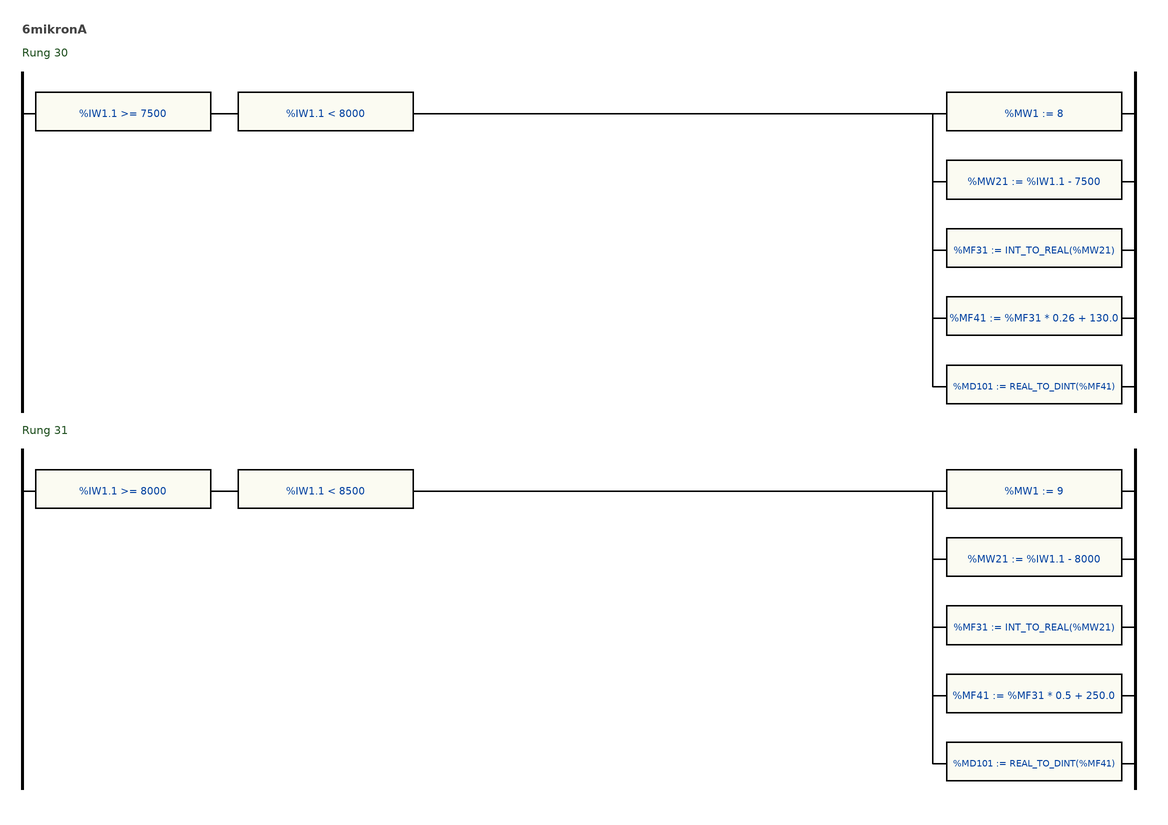

// Rung 30
  LD [ %IW1.1 >= 7500 ]
  AND [ %IW1.1 < 8000 ]
  [ %MW1 := 8 ]
  [ %MW21 := %IW1.1 - 7500 ]
  [ %MF31 := INT_TO_REAL ( %MW21 ) ]
  [ %MF41 := %MF31 * 0.26 + 130.0 ]
  [ %MD101 := REAL_TO_DINT ( %MF41 ) ]
  // as ST:
  //   IF %IW1.1 >= 7500 AND %IW1.1 < 8000 THEN %MW1 := 8; END_IF;
  //   IF %IW1.1 >= 7500 AND %IW1.1 < 8000 THEN %MW21 := %IW1.1 - 7500; END_IF;
  //   IF %IW1.1 >= 7500 AND %IW1.1 < 8000 THEN %MF31 := INT_TO_REAL ( %MW21 ); END_IF;
  //   IF %IW1.1 >= 7500 AND %IW1.1 < 8000 THEN %MF41 := %MF31 * 0.26 + 130.0; END_IF;
  //   IF %IW1.1 >= 7500 AND %IW1.1 < 8000 THEN %MD101 := REAL_TO_DINT ( %MF41 ); END_IF;

// Rung 31
  LD [ %IW1.1 >= 8000 ]
  AND [ %IW1.1 < 8500 ]
  [ %MW1 := 9 ]
  [ %MW21 := %IW1.1 - 8000 ]
  [ %MF31 := INT_TO_REAL ( %MW21 ) ]
  [ %MF41 := %MF31 * 0.5 + 250.0 ]
  [ %MD101 := REAL_TO_DINT ( %MF41 ) ]
  // as ST:
  //   IF %IW1.1 >= 8000 AND %IW1.1 < 8500 THEN %MW1 := 9; END_IF;
  //   IF %IW1.1 >= 8000 AND %IW1.1 < 8500 THEN %MW21 := %IW1.1 - 8000; END_IF;
  //   IF %IW1.1 >= 8000 AND %IW1.1 < 8500 THEN %MF31 := INT_TO_REAL ( %MW21 ); END_IF;
  //   IF %IW1.1 >= 8000 AND %IW1.1 < 8500 THEN %MF41 := %MF31 * 0.5 + 250.0; END_IF;
  //   IF %IW1.1 >= 8000 AND %IW1.1 < 8500 THEN %MD101 := REAL_TO_DINT ( %MF41 ); END_IF;

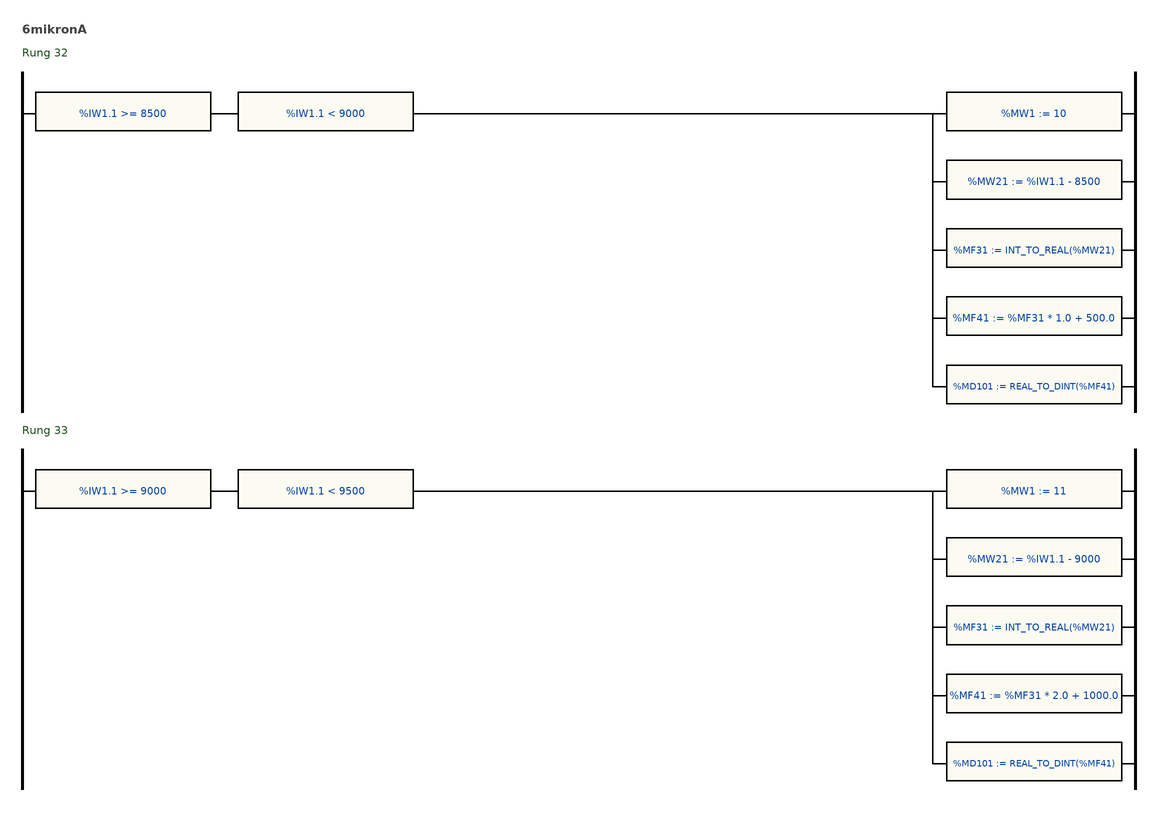

// Rung 32
  LD [ %IW1.1 >= 8500 ]
  AND [ %IW1.1 < 9000 ]
  [ %MW1 := 10 ]
  [ %MW21 := %IW1.1 - 8500 ]
  [ %MF31 := INT_TO_REAL ( %MW21 ) ]
  [ %MF41 := %MF31 * 1.0 + 500.0 ]
  [ %MD101 := REAL_TO_DINT ( %MF41 ) ]
  // as ST:
  //   IF %IW1.1 >= 8500 AND %IW1.1 < 9000 THEN %MW1 := 10; END_IF;
  //   IF %IW1.1 >= 8500 AND %IW1.1 < 9000 THEN %MW21 := %IW1.1 - 8500; END_IF;
  //   IF %IW1.1 >= 8500 AND %IW1.1 < 9000 THEN %MF31 := INT_TO_REAL ( %MW21 ); END_IF;
  //   IF %IW1.1 >= 8500 AND %IW1.1 < 9000 THEN %MF41 := %MF31 * 1.0 + 500.0; END_IF;
  //   IF %IW1.1 >= 8500 AND %IW1.1 < 9000 THEN %MD101 := REAL_TO_DINT ( %MF41 ); END_IF;

// Rung 33
  LD [ %IW1.1 >= 9000 ]
  AND [ %IW1.1 < 9500 ]
  [ %MW1 := 11 ]
  [ %MW21 := %IW1.1 - 9000 ]
  [ %MF31 := INT_TO_REAL ( %MW21 ) ]
  [ %MF41 := %MF31 * 2.0 + 1000.0 ]
  [ %MD101 := REAL_TO_DINT ( %MF41 ) ]
  // as ST:
  //   IF %IW1.1 >= 9000 AND %IW1.1 < 9500 THEN %MW1 := 11; END_IF;
  //   IF %IW1.1 >= 9000 AND %IW1.1 < 9500 THEN %MW21 := %IW1.1 - 9000; END_IF;
  //   IF %IW1.1 >= 9000 AND %IW1.1 < 9500 THEN %MF31 := INT_TO_REAL ( %MW21 ); END_IF;
  //   IF %IW1.1 >= 9000 AND %IW1.1 < 9500 THEN %MF41 := %MF31 * 2.0 + 1000.0; END_IF;
  //   IF %IW1.1 >= 9000 AND %IW1.1 < 9500 THEN %MD101 := REAL_TO_DINT ( %MF41 ); END_IF;

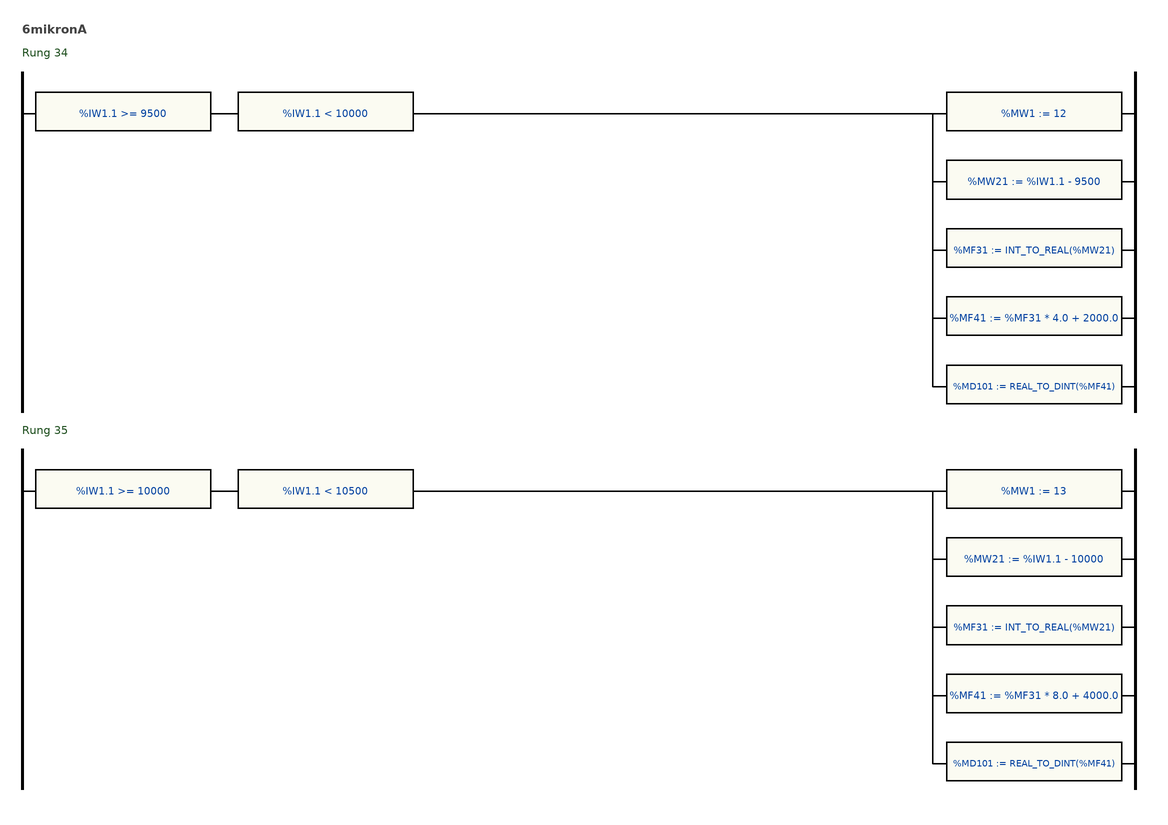

// Rung 34
  LD [ %IW1.1 >= 9500 ]
  AND [ %IW1.1 < 10000 ]
  [ %MW1 := 12 ]
  [ %MW21 := %IW1.1 - 9500 ]
  [ %MF31 := INT_TO_REAL ( %MW21 ) ]
  [ %MF41 := %MF31 * 4.0 + 2000.0 ]
  [ %MD101 := REAL_TO_DINT ( %MF41 ) ]
  // as ST:
  //   IF %IW1.1 >= 9500 AND %IW1.1 < 10000 THEN %MW1 := 12; END_IF;
  //   IF %IW1.1 >= 9500 AND %IW1.1 < 10000 THEN %MW21 := %IW1.1 - 9500; END_IF;
  //   IF %IW1.1 >= 9500 AND %IW1.1 < 10000 THEN %MF31 := INT_TO_REAL ( %MW21 ); END_IF;
  //   IF %IW1.1 >= 9500 AND %IW1.1 < 10000 THEN %MF41 := %MF31 * 4.0 + 2000.0; END_IF;
  //   IF %IW1.1 >= 9500 AND %IW1.1 < 10000 THEN %MD101 := REAL_TO_DINT ( %MF41 ); END_IF;

// Rung 35
  LD [ %IW1.1 >= 10000 ]
  AND [ %IW1.1 < 10500 ]
  [ %MW1 := 13 ]
  [ %MW21 := %IW1.1 - 10000 ]
  [ %MF31 := INT_TO_REAL ( %MW21 ) ]
  [ %MF41 := %MF31 * 8.0 + 4000.0 ]
  [ %MD101 := REAL_TO_DINT ( %MF41 ) ]
  // as ST:
  //   IF %IW1.1 >= 10000 AND %IW1.1 < 10500 THEN %MW1 := 13; END_IF;
  //   IF %IW1.1 >= 10000 AND %IW1.1 < 10500 THEN %MW21 := %IW1.1 - 10000; END_IF;
  //   IF %IW1.1 >= 10000 AND %IW1.1 < 10500 THEN %MF31 := INT_TO_REAL ( %MW21 ); END_IF;
  //   IF %IW1.1 >= 10000 AND %IW1.1 < 10500 THEN %MF41 := %MF31 * 8.0 + 4000.0; END_IF;
  //   IF %IW1.1 >= 10000 AND %IW1.1 < 10500 THEN %MD101 := REAL_TO_DINT ( %MF41 ); END_IF;

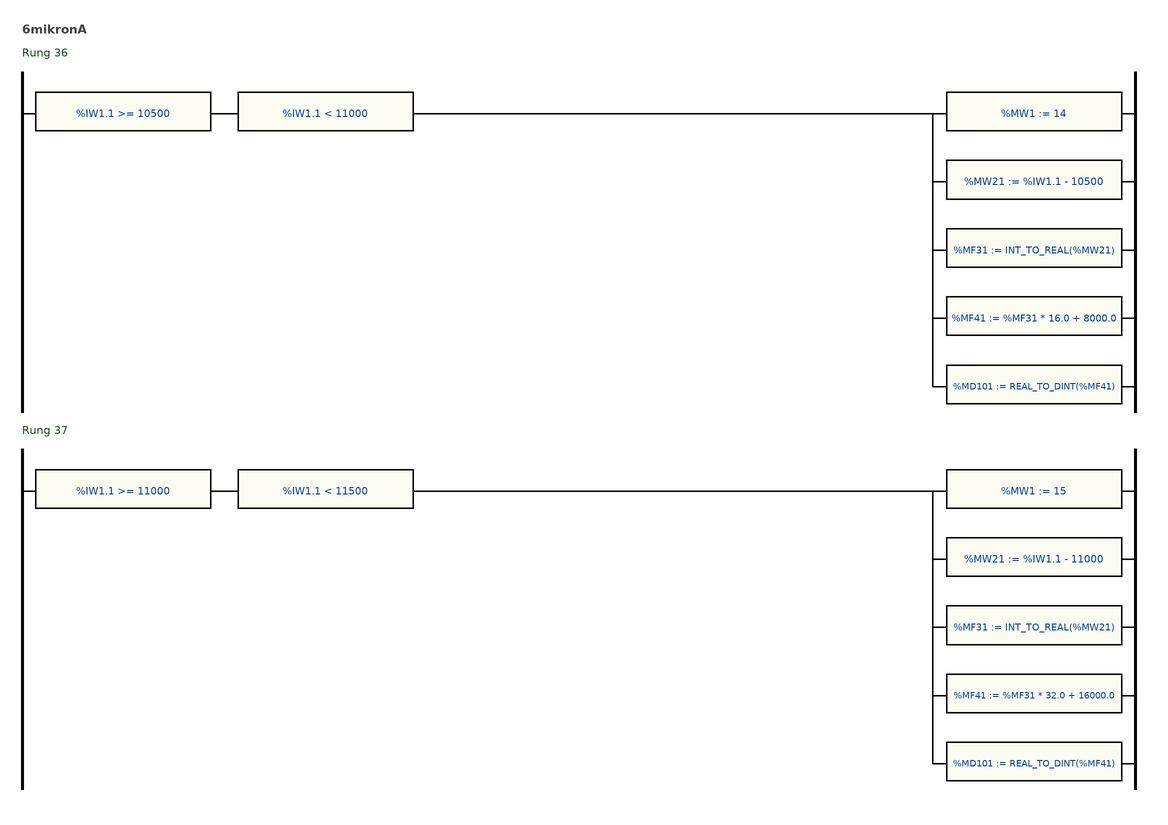

// Rung 36
  LD [ %IW1.1 >= 10500 ]
  AND [ %IW1.1 < 11000 ]
  [ %MW1 := 14 ]
  [ %MW21 := %IW1.1 - 10500 ]
  [ %MF31 := INT_TO_REAL ( %MW21 ) ]
  [ %MF41 := %MF31 * 16.0 + 8000.0 ]
  [ %MD101 := REAL_TO_DINT ( %MF41 ) ]
  // as ST:
  //   IF %IW1.1 >= 10500 AND %IW1.1 < 11000 THEN %MW1 := 14; END_IF;
  //   IF %IW1.1 >= 10500 AND %IW1.1 < 11000 THEN %MW21 := %IW1.1 - 10500; END_IF;
  //   IF %IW1.1 >= 10500 AND %IW1.1 < 11000 THEN %MF31 := INT_TO_REAL ( %MW21 ); END_IF;
  //   IF %IW1.1 >= 10500 AND %IW1.1 < 11000 THEN %MF41 := %MF31 * 16.0 + 8000.0; END_IF;
  //   IF %IW1.1 >= 10500 AND %IW1.1 < 11000 THEN %MD101 := REAL_TO_DINT ( %MF41 ); END_IF;

// Rung 37
  LD [ %IW1.1 >= 11000 ]
  AND [ %IW1.1 < 11500 ]
  [ %MW1 := 15 ]
  [ %MW21 := %IW1.1 - 11000 ]
  [ %MF31 := INT_TO_REAL ( %MW21 ) ]
  [ %MF41 := %MF31 * 32.0 + 16000.0 ]
  [ %MD101 := REAL_TO_DINT ( %MF41 ) ]
  // as ST:
  //   IF %IW1.1 >= 11000 AND %IW1.1 < 11500 THEN %MW1 := 15; END_IF;
  //   IF %IW1.1 >= 11000 AND %IW1.1 < 11500 THEN %MW21 := %IW1.1 - 11000; END_IF;
  //   IF %IW1.1 >= 11000 AND %IW1.1 < 11500 THEN %MF31 := INT_TO_REAL ( %MW21 ); END_IF;
  //   IF %IW1.1 >= 11000 AND %IW1.1 < 11500 THEN %MF41 := %MF31 * 32.0 + 16000.0; END_IF;
  //   IF %IW1.1 >= 11000 AND %IW1.1 < 11500 THEN %MD101 := REAL_TO_DINT ( %MF41 ); END_IF;

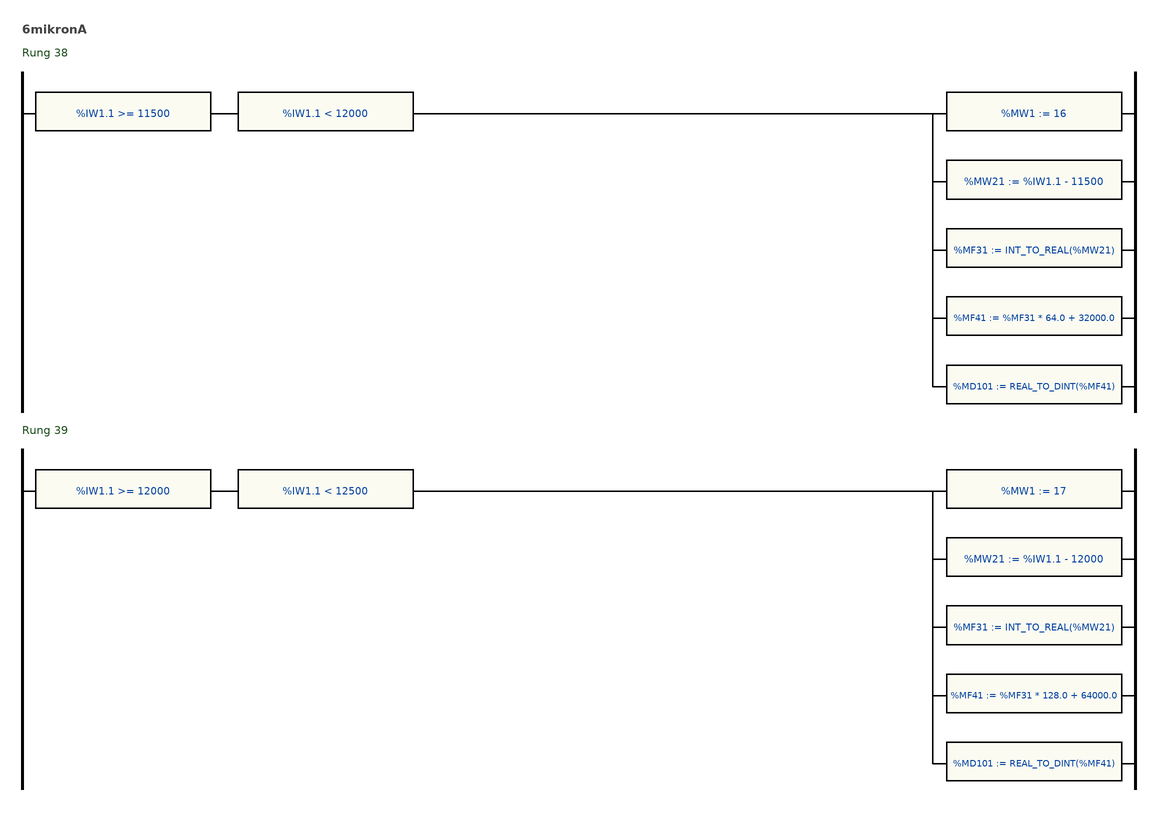

// Rung 38
  LD [ %IW1.1 >= 11500 ]
  AND [ %IW1.1 < 12000 ]
  [ %MW1 := 16 ]
  [ %MW21 := %IW1.1 - 11500 ]
  [ %MF31 := INT_TO_REAL ( %MW21 ) ]
  [ %MF41 := %MF31 * 64.0 + 32000.0 ]
  [ %MD101 := REAL_TO_DINT ( %MF41 ) ]
  // as ST:
  //   IF %IW1.1 >= 11500 AND %IW1.1 < 12000 THEN %MW1 := 16; END_IF;
  //   IF %IW1.1 >= 11500 AND %IW1.1 < 12000 THEN %MW21 := %IW1.1 - 11500; END_IF;
  //   IF %IW1.1 >= 11500 AND %IW1.1 < 12000 THEN %MF31 := INT_TO_REAL ( %MW21 ); END_IF;
  //   IF %IW1.1 >= 11500 AND %IW1.1 < 12000 THEN %MF41 := %MF31 * 64.0 + 32000.0; END_IF;
  //   IF %IW1.1 >= 11500 AND %IW1.1 < 12000 THEN %MD101 := REAL_TO_DINT ( %MF41 ); END_IF;

// Rung 39
  LD [ %IW1.1 >= 12000 ]
  AND [ %IW1.1 < 12500 ]
  [ %MW1 := 17 ]
  [ %MW21 := %IW1.1 - 12000 ]
  [ %MF31 := INT_TO_REAL ( %MW21 ) ]
  [ %MF41 := %MF31 * 128.0 + 64000.0 ]
  [ %MD101 := REAL_TO_DINT ( %MF41 ) ]
  // as ST:
  //   IF %IW1.1 >= 12000 AND %IW1.1 < 12500 THEN %MW1 := 17; END_IF;
  //   IF %IW1.1 >= 12000 AND %IW1.1 < 12500 THEN %MW21 := %IW1.1 - 12000; END_IF;
  //   IF %IW1.1 >= 12000 AND %IW1.1 < 12500 THEN %MF31 := INT_TO_REAL ( %MW21 ); END_IF;
  //   IF %IW1.1 >= 12000 AND %IW1.1 < 12500 THEN %MF41 := %MF31 * 128.0 + 64000.0; END_IF;
  //   IF %IW1.1 >= 12000 AND %IW1.1 < 12500 THEN %MD101 := REAL_TO_DINT ( %MF41 ); END_IF;

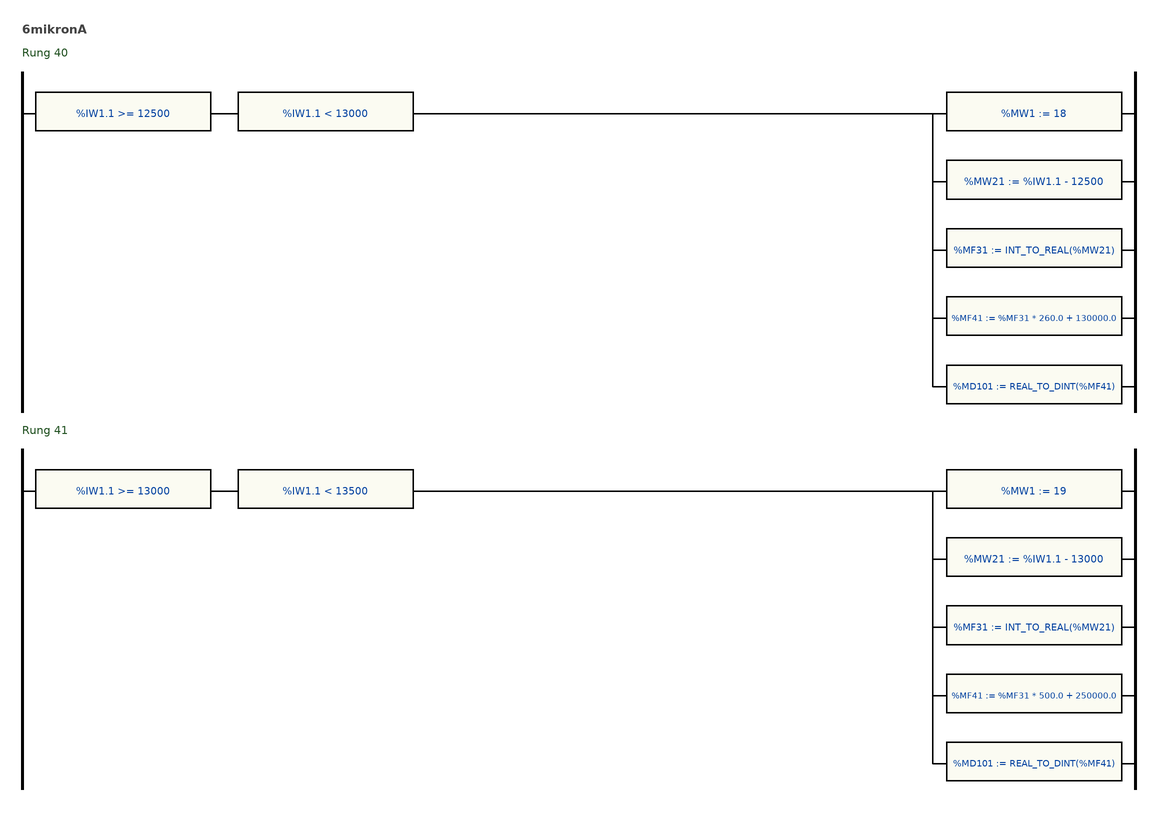

// Rung 40
  LD [ %IW1.1 >= 12500 ]
  AND [ %IW1.1 < 13000 ]
  [ %MW1 := 18 ]
  [ %MW21 := %IW1.1 - 12500 ]
  [ %MF31 := INT_TO_REAL ( %MW21 ) ]
  [ %MF41 := %MF31 * 260.0 + 130000.0 ]
  [ %MD101 := REAL_TO_DINT ( %MF41 ) ]
  // as ST:
  //   IF %IW1.1 >= 12500 AND %IW1.1 < 13000 THEN %MW1 := 18; END_IF;
  //   IF %IW1.1 >= 12500 AND %IW1.1 < 13000 THEN %MW21 := %IW1.1 - 12500; END_IF;
  //   IF %IW1.1 >= 12500 AND %IW1.1 < 13000 THEN %MF31 := INT_TO_REAL ( %MW21 ); END_IF;
  //   IF %IW1.1 >= 12500 AND %IW1.1 < 13000 THEN %MF41 := %MF31 * 260.0 + 130000.0; END_IF;
  //   IF %IW1.1 >= 12500 AND %IW1.1 < 13000 THEN %MD101 := REAL_TO_DINT ( %MF41 ); END_IF;

// Rung 41
  LD [ %IW1.1 >= 13000 ]
  AND [ %IW1.1 < 13500 ]
  [ %MW1 := 19 ]
  [ %MW21 := %IW1.1 - 13000 ]
  [ %MF31 := INT_TO_REAL ( %MW21 ) ]
  [ %MF41 := %MF31 * 500.0 + 250000.0 ]
  [ %MD101 := REAL_TO_DINT ( %MF41 ) ]
  // as ST:
  //   IF %IW1.1 >= 13000 AND %IW1.1 < 13500 THEN %MW1 := 19; END_IF;
  //   IF %IW1.1 >= 13000 AND %IW1.1 < 13500 THEN %MW21 := %IW1.1 - 13000; END_IF;
  //   IF %IW1.1 >= 13000 AND %IW1.1 < 13500 THEN %MF31 := INT_TO_REAL ( %MW21 ); END_IF;
  //   IF %IW1.1 >= 13000 AND %IW1.1 < 13500 THEN %MF41 := %MF31 * 500.0 + 250000.0; END_IF;
  //   IF %IW1.1 >= 13000 AND %IW1.1 < 13500 THEN %MD101 := REAL_TO_DINT ( %MF41 ); END_IF;

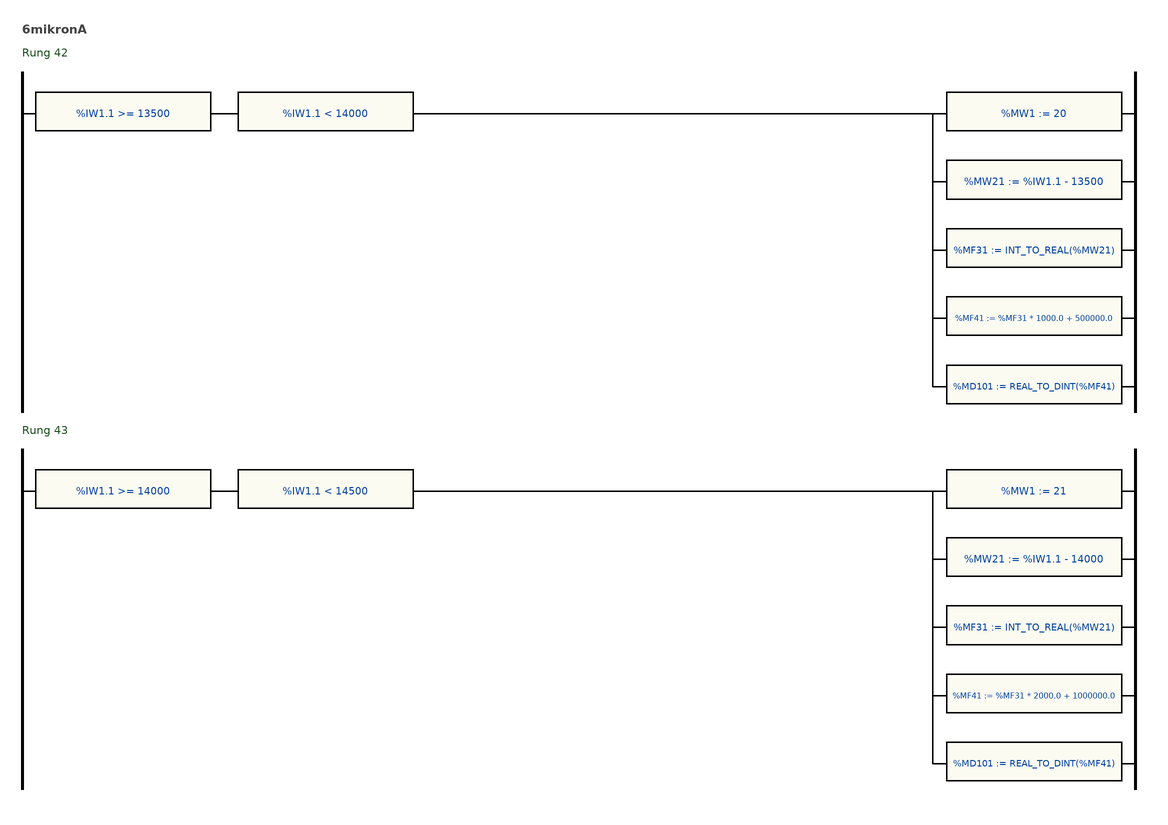

// Rung 42
  LD [ %IW1.1 >= 13500 ]
  AND [ %IW1.1 < 14000 ]
  [ %MW1 := 20 ]
  [ %MW21 := %IW1.1 - 13500 ]
  [ %MF31 := INT_TO_REAL ( %MW21 ) ]
  [ %MF41 := %MF31 * 1000.0 + 500000.0 ]
  [ %MD101 := REAL_TO_DINT ( %MF41 ) ]
  // as ST:
  //   IF %IW1.1 >= 13500 AND %IW1.1 < 14000 THEN %MW1 := 20; END_IF;
  //   IF %IW1.1 >= 13500 AND %IW1.1 < 14000 THEN %MW21 := %IW1.1 - 13500; END_IF;
  //   IF %IW1.1 >= 13500 AND %IW1.1 < 14000 THEN %MF31 := INT_TO_REAL ( %MW21 ); END_IF;
  //   IF %IW1.1 >= 13500 AND %IW1.1 < 14000 THEN %MF41 := %MF31 * 1000.0 + 500000.0; END_IF;
  //   IF %IW1.1 >= 13500 AND %IW1.1 < 14000 THEN %MD101 := REAL_TO_DINT ( %MF41 ); END_IF;

// Rung 43
  LD [ %IW1.1 >= 14000 ]
  AND [ %IW1.1 < 14500 ]
  [ %MW1 := 21 ]
  [ %MW21 := %IW1.1 - 14000 ]
  [ %MF31 := INT_TO_REAL ( %MW21 ) ]
  [ %MF41 := %MF31 * 2000.0 + 1000000.0 ]
  [ %MD101 := REAL_TO_DINT ( %MF41 ) ]
  // as ST:
  //   IF %IW1.1 >= 14000 AND %IW1.1 < 14500 THEN %MW1 := 21; END_IF;
  //   IF %IW1.1 >= 14000 AND %IW1.1 < 14500 THEN %MW21 := %IW1.1 - 14000; END_IF;
  //   IF %IW1.1 >= 14000 AND %IW1.1 < 14500 THEN %MF31 := INT_TO_REAL ( %MW21 ); END_IF;
  //   IF %IW1.1 >= 14000 AND %IW1.1 < 14500 THEN %MF41 := %MF31 * 2000.0 + 1000000.0; END_IF;
  //   IF %IW1.1 >= 14000 AND %IW1.1 < 14500 THEN %MD101 := REAL_TO_DINT ( %MF41 ); END_IF;

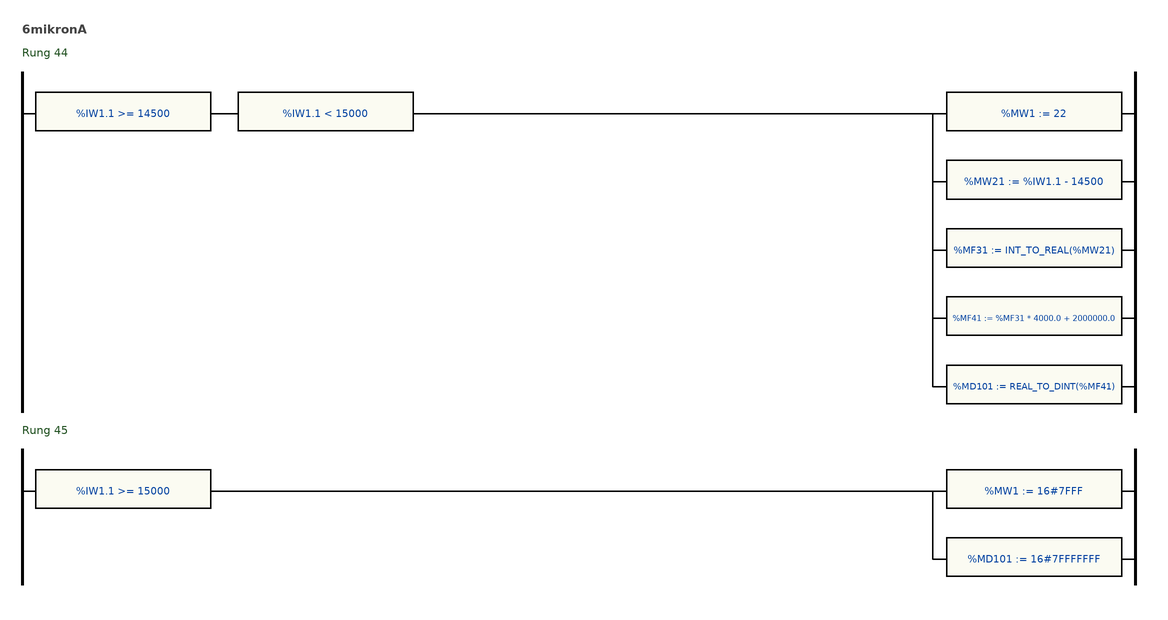

// Rung 44
  LD [ %IW1.1 >= 14500 ]
  AND [ %IW1.1 < 15000 ]
  [ %MW1 := 22 ]
  [ %MW21 := %IW1.1 - 14500 ]
  [ %MF31 := INT_TO_REAL ( %MW21 ) ]
  [ %MF41 := %MF31 * 4000.0 + 2000000.0 ]
  [ %MD101 := REAL_TO_DINT ( %MF41 ) ]
  // as ST:
  //   IF %IW1.1 >= 14500 AND %IW1.1 < 15000 THEN %MW1 := 22; END_IF;
  //   IF %IW1.1 >= 14500 AND %IW1.1 < 15000 THEN %MW21 := %IW1.1 - 14500; END_IF;
  //   IF %IW1.1 >= 14500 AND %IW1.1 < 15000 THEN %MF31 := INT_TO_REAL ( %MW21 ); END_IF;
  //   IF %IW1.1 >= 14500 AND %IW1.1 < 15000 THEN %MF41 := %MF31 * 4000.0 + 2000000.0; END_IF;
  //   IF %IW1.1 >= 14500 AND %IW1.1 < 15000 THEN %MD101 := REAL_TO_DINT ( %MF41 ); END_IF;

// Rung 45
  LD [ %IW1.1 >= 15000 ]
  [ %MW1 := 16#7FFF ]
  [ %MD101 := 16#7FFFFFFF ]
  // as ST:
  //   IF %IW1.1 >= 15000 THEN %MW1 := 16#7FFF; END_IF;
  //   IF %IW1.1 >= 15000 THEN %MD101 := 16#7FFFFFFF; END_IF;

POU 14mikronA
  (* SectionNumber=3 *)

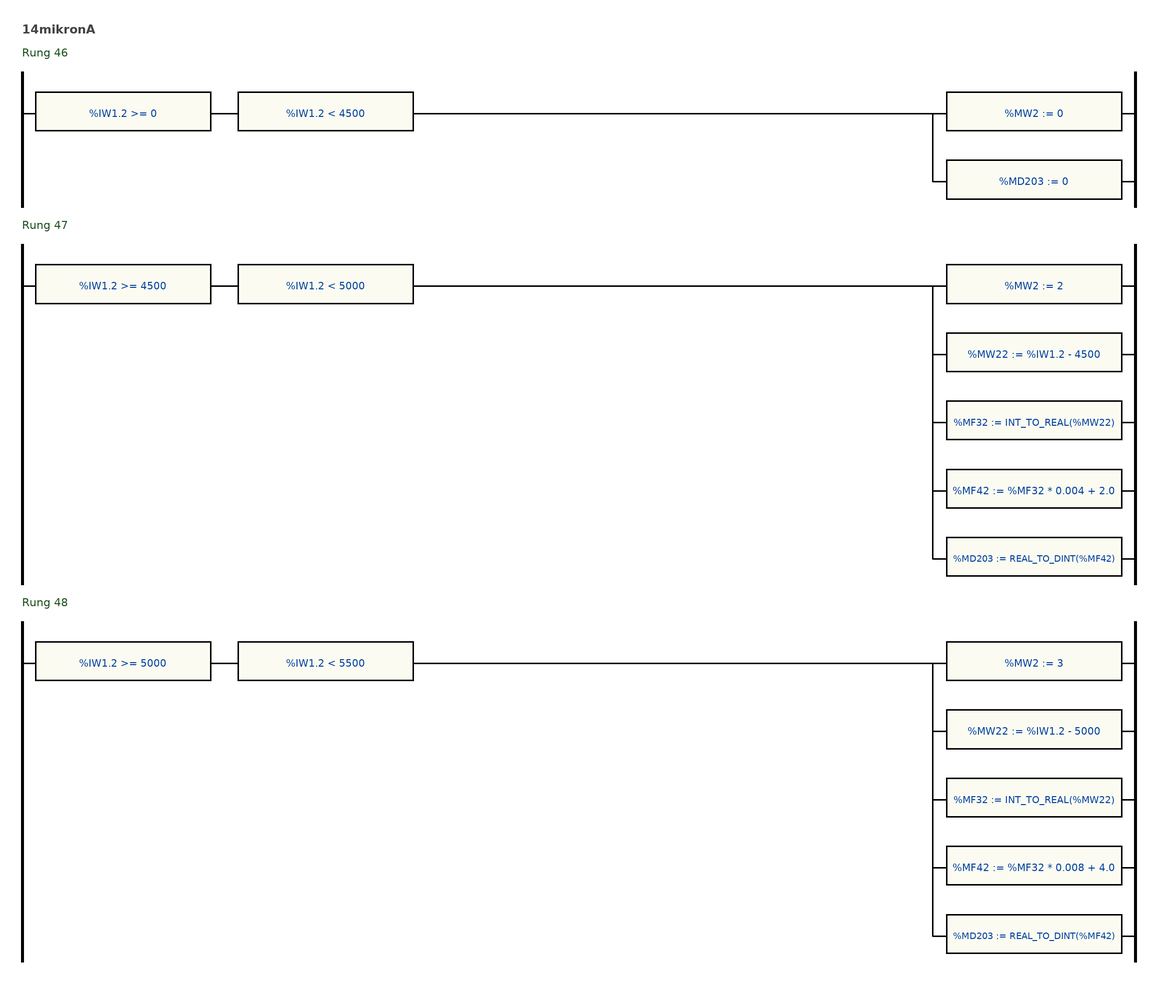

// Rung 46
  LD [ %IW1.2 >= 0 ]
  AND [ %IW1.2 < 4500 ]
  [ %MW2 := 0 ]
  [ %MD203 := 0 ]
  // as ST:
  //   IF %IW1.2 >= 0 AND %IW1.2 < 4500 THEN %MW2 := 0; END_IF;
  //   IF %IW1.2 >= 0 AND %IW1.2 < 4500 THEN %MD203 := 0; END_IF;

// Rung 47
  LD [ %IW1.2 >= 4500 ]
  AND [ %IW1.2 < 5000 ]
  [ %MW2 := 2 ]
  [ %MW22 := %IW1.2 - 4500 ]
  [ %MF32 := INT_TO_REAL ( %MW22 ) ]
  [ %MF42 := %MF32 * 0.004 + 2.0 ]
  [ %MD203 := REAL_TO_DINT ( %MF42 ) ]
  // as ST:
  //   IF %IW1.2 >= 4500 AND %IW1.2 < 5000 THEN %MW2 := 2; END_IF;
  //   IF %IW1.2 >= 4500 AND %IW1.2 < 5000 THEN %MW22 := %IW1.2 - 4500; END_IF;
  //   IF %IW1.2 >= 4500 AND %IW1.2 < 5000 THEN %MF32 := INT_TO_REAL ( %MW22 ); END_IF;
  //   IF %IW1.2 >= 4500 AND %IW1.2 < 5000 THEN %MF42 := %MF32 * 0.004 + 2.0; END_IF;
  //   IF %IW1.2 >= 4500 AND %IW1.2 < 5000 THEN %MD203 := REAL_TO_DINT ( %MF42 ); END_IF;

// Rung 48
  LD [ %IW1.2 >= 5000 ]
  AND [ %IW1.2 < 5500 ]
  [ %MW2 := 3 ]
  [ %MW22 := %IW1.2 - 5000 ]
  [ %MF32 := INT_TO_REAL ( %MW22 ) ]
  [ %MF42 := %MF32 * 0.008 + 4.0 ]
  [ %MD203 := REAL_TO_DINT ( %MF42 ) ]
  // as ST:
  //   IF %IW1.2 >= 5000 AND %IW1.2 < 5500 THEN %MW2 := 3; END_IF;
  //   IF %IW1.2 >= 5000 AND %IW1.2 < 5500 THEN %MW22 := %IW1.2 - 5000; END_IF;
  //   IF %IW1.2 >= 5000 AND %IW1.2 < 5500 THEN %MF32 := INT_TO_REAL ( %MW22 ); END_IF;
  //   IF %IW1.2 >= 5000 AND %IW1.2 < 5500 THEN %MF42 := %MF32 * 0.008 + 4.0; END_IF;
  //   IF %IW1.2 >= 5000 AND %IW1.2 < 5500 THEN %MD203 := REAL_TO_DINT ( %MF42 ); END_IF;

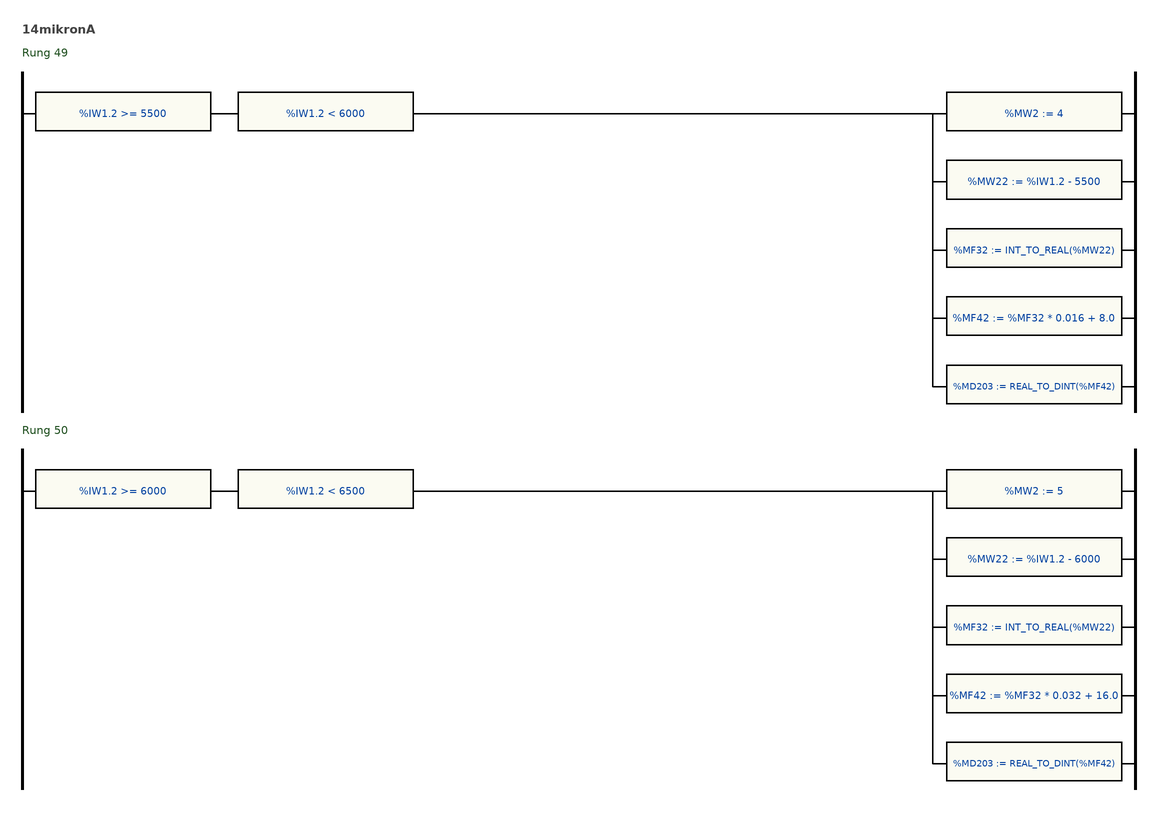

// Rung 49
  LD [ %IW1.2 >= 5500 ]
  AND [ %IW1.2 < 6000 ]
  [ %MW2 := 4 ]
  [ %MW22 := %IW1.2 - 5500 ]
  [ %MF32 := INT_TO_REAL ( %MW22 ) ]
  [ %MF42 := %MF32 * 0.016 + 8.0 ]
  [ %MD203 := REAL_TO_DINT ( %MF42 ) ]
  // as ST:
  //   IF %IW1.2 >= 5500 AND %IW1.2 < 6000 THEN %MW2 := 4; END_IF;
  //   IF %IW1.2 >= 5500 AND %IW1.2 < 6000 THEN %MW22 := %IW1.2 - 5500; END_IF;
  //   IF %IW1.2 >= 5500 AND %IW1.2 < 6000 THEN %MF32 := INT_TO_REAL ( %MW22 ); END_IF;
  //   IF %IW1.2 >= 5500 AND %IW1.2 < 6000 THEN %MF42 := %MF32 * 0.016 + 8.0; END_IF;
  //   IF %IW1.2 >= 5500 AND %IW1.2 < 6000 THEN %MD203 := REAL_TO_DINT ( %MF42 ); END_IF;

// Rung 50
  LD [ %IW1.2 >= 6000 ]
  AND [ %IW1.2 < 6500 ]
  [ %MW2 := 5 ]
  [ %MW22 := %IW1.2 - 6000 ]
  [ %MF32 := INT_TO_REAL ( %MW22 ) ]
  [ %MF42 := %MF32 * 0.032 + 16.0 ]
  [ %MD203 := REAL_TO_DINT ( %MF42 ) ]
  // as ST:
  //   IF %IW1.2 >= 6000 AND %IW1.2 < 6500 THEN %MW2 := 5; END_IF;
  //   IF %IW1.2 >= 6000 AND %IW1.2 < 6500 THEN %MW22 := %IW1.2 - 6000; END_IF;
  //   IF %IW1.2 >= 6000 AND %IW1.2 < 6500 THEN %MF32 := INT_TO_REAL ( %MW22 ); END_IF;
  //   IF %IW1.2 >= 6000 AND %IW1.2 < 6500 THEN %MF42 := %MF32 * 0.032 + 16.0; END_IF;
  //   IF %IW1.2 >= 6000 AND %IW1.2 < 6500 THEN %MD203 := REAL_TO_DINT ( %MF42 ); END_IF;

